LIN {X 0,Y 377.924,Z 388.108,A -85,B 0,C 180,E1 -14679.457,E2 -14679.457} C_VEL
LIN {X 0,Y 374.794,Z 386.154,A -85,B 0,C 180,E1 -14680.722,E2 -14680.722} C_VEL
LIN {X 0,Y 371.596,Z 383.295,A -85,B 0,C 180,E1 -14681.935,E2 -14681.935} C_VEL
LIN {X 0,Y 368.955,Z 380.545,A -85,B 0,C 180,E1 -14682.86,E2 -14682.86} C_VEL
LIN {X 0,Y 365.594,Z 377.85,A -85,B 0,C 180,E1 -14683.883,E2 -14683.883} C_VEL
LIN {X 0,Y 361.342,Z 373.442,A -85,B 0,C 180,E1 -14685.107,E2 -14685.107} C_VEL
LIN {X 0,Y 357.377,Z 369.827,A -85,B 0,C 180,E1 -14686.133,E2 -14686.133} C_VEL
LIN {X 0,Y 354.406,Z 366.631,A -85,B 0,C 180,E1 -14686.847,E2 -14686.847} C_VEL
LIN {X 0,Y 350.901,Z 363.042,A -85,B 0,C 180,E1 -14687.655,E2 -14687.655} C_VEL
LIN {X 0,Y 348.553,Z 360.395,A -85,B 0,C 180,E1 -14688.184,E2 -14688.184} C_VEL
LIN {X 0,Y 345.155,Z 356.37,A -85,B 0,C 180,E1 -14688.921,E2 -14688.921} C_VEL
LIN {X 0,Y 341.007,Z 351.456,A -85,B 0,C 180,E1 -14689.766,E2 -14689.766} C_VEL
LIN {X 0,Y 339.565,Z 349.602,A -85,B 0,C 180,E1 -14690.055,E2 -14690.055} C_VEL
LIN {X 0,Y 337.185,Z 346.417,A -85,B 0,C 180,E1 -14690.522,E2 -14690.522} C_VEL
LIN {X 0,Y 336.133,Z 344.943,A -85,B 0,C 180,E1 -14690.724,E2 -14690.724} C_VEL
LIN {X 0,Y 334.263,Z 342.48,A -85,B 0,C 180,E1 -14691.08,E2 -14691.08} C_VEL
LIN {X 0,Y 333.682,Z 340.419,A -85,B 0,C 180,E1 -14691.257,E2 -14691.257} C_VEL
LIN {X 0,Y 333.715,Z 340.414,A -85,B 0,C 180,E1 -14695.101,E2 -14695.101} C_VEL
LIN {X 0,Y 333.717,Z 340.415,A -85,B 0,C 180,E1 -14697.811,E2 -14697.811} C_VEL
LIN {X 0,Y 333.693,Z 340.421,A -85,B 0,C 180,E1 -14700.362,E2 -14700.362} C_VEL
LIN {X 0,Y 333.67,Z 340.42,A -85,B 0,C 180,E1 -14704.659,E2 -14704.659} C_VEL
LIN {X 0,Y 333.652,Z 340.423,A -85,B 0,C 180,E1 -14707.651,E2 -14707.651} C_VEL
LIN {X 0,Y 333.652,Z 340.421,A -85,B 0,C 180,E1 -14710.766,E2 -14710.766} C_VEL
LIN {X 0,Y 333.659,Z 340.422,A -85,B 0,C 180,E1 -14714.263,E2 -14714.263} C_VEL
LIN {X 0,Y 333.693,Z 340.419,A -85,B 0,C 180,E1 -14717.627,E2 -14717.627} C_VEL
LIN {X 0,Y 333.679,Z 340.419,A -85,B 0,C 180,E1 -14721.196,E2 -14721.196} C_VEL
LIN {X 0,Y 333.682,Z 340.419,A -85,B 0,C 180,E1 -14725.226,E2 -14725.226} C_VEL
LIN {X 0,Y 333.631,Z 340.424,A -85,B 0,C 180,E1 -14728.223,E2 -14728.223} C_VEL
LIN {X 0,Y 333.708,Z 340.415,A -85,B 0,C 180,E1 -14731.029,E2 -14731.029} C_VEL
LIN {X 0,Y 333.709,Z 340.413,A -85,B 0,C 180,E1 -14734.677,E2 -14734.677} C_VEL
LIN {X 0,Y 333.662,Z 340.421,A -85,B 0,C 180,E1 -14737.938,E2 -14737.938} C_VEL
LIN {X 0,Y 333.696,Z 340.413,A -85,B 0,C 180,E1 -14739.91,E2 -14739.91} C_VEL
LIN {X 0,Y 333.087,Z 340.494,A -85,B 0,C 180,E1 -14740.917,E2 -14740.917} C_VEL
LIN {X 0,Y 330.266,Z 340.846,A -85,B 0,C 180,E1 -14742.557,E2 -14742.557} C_VEL
LIN {X 0,Y 327.852,Z 341.148,A -85,B 0,C 180,E1 -14743.884,E2 -14743.884} C_VEL
LIN {X 0,Y 326.829,Z 341.275,A -85,B 0,C 180,E1 -14744.912,E2 -14744.912} C_VEL
LIN {X 0,Y 326.756,Z 341.283,A -85,B 0,C 180,E1 -14745.26,E2 -14745.26} C_VEL
LIN {X 0,Y 326.768,Z 341.282,A -85,B 0,C 180,E1 -14748.84,E2 -14748.84} C_VEL
LIN {X 0,Y 326.965,Z 341.256,A -85,B 0,C 180,E1 -14752.591,E2 -14752.591} C_VEL
LIN {X 0,Y 326.775,Z 341.28,A -85,B 0,C 180,E1 -14755.066,E2 -14755.066} C_VEL
LIN {X 0,Y 327.047,Z 341.239,A -85,B 0,C 180,E1 -14757.537,E2 -14757.537} C_VEL
LIN {X 0,Y 327.178,Z 341.224,A -85,B 0,C 180,E1 -14760.001,E2 -14760.001} C_VEL
LIN {X 0,Y 327.046,Z 341.246,A -85,B 0,C 180,E1 -14762.464,E2 -14762.464} C_VEL
LIN {X 0,Y 326.989,Z 341.252,A -85,B 0,C 180,E1 -14766.17,E2 -14766.17} C_VEL
LIN {X 0,Y 326.914,Z 341.266,A -85,B 0,C 180,E1 -14768.656,E2 -14768.656} C_VEL
LIN {X 0,Y 326.735,Z 341.288,A -85,B 0,C 180,E1 -14772.422,E2 -14772.422} C_VEL
LIN {X 0,Y 326.751,Z 341.283,A -85,B 0,C 180,E1 -14774.958,E2 -14774.958} C_VEL
LIN {X 0,Y 326.707,Z 341.288,A -85,B 0,C 180,E1 -14778.825,E2 -14778.825} C_VEL
LIN {X 0,Y 326.603,Z 341.301,A -85,B 0,C 180,E1 -14782.789,E2 -14782.789} C_VEL
LIN {X 0,Y 326.69,Z 341.29,A -85,B 0,C 180,E1 -14785.484,E2 -14785.484} C_VEL
LIN {X 0,Y 326.649,Z 341.296,A -85,B 0,C 180,E1 -14789.661,E2 -14789.661} C_VEL
LIN {X 0,Y 326.608,Z 341.305,A -85,B 0,C 180,E1 -14794.02,E2 -14794.02} C_VEL
LIN {X 0,Y 326.687,Z 341.65,A -85,B 0,C 180,E1 -14795.511,E2 -14795.511} C_VEL
LIN {X 0,Y 327.029,Z 344.299,A -85,B 0,C 180,E1 -14799.317,E2 -14799.317} C_VEL
LIN {X 0,Y 327.299,Z 346.11,A -85,B 0,C 180,E1 -14801.733,E2 -14801.733} C_VEL
LIN {X 0,Y 327.621,Z 348.814,A -85,B 0,C 180,E1 -14805.065,E2 -14805.065} C_VEL
LIN {X 0,Y 327.642,Z 351.691,A -85,B 0,C 180,E1 -14808.321,E2 -14808.321} C_VEL
LIN {X 0,Y 327.31,Z 354.713,A -85,B 0,C 180,E1 -14811.488,E2 -14811.488} C_VEL
LIN {X 0,Y 326.873,Z 358.059,A -85,B 0,C 180,E1 -14814.789,E2 -14814.789} C_VEL
LIN {X 0,Y 326.311,Z 362.418,A -85,B 0,C 180,E1 -14818.875,E2 -14818.875} C_VEL
LIN {X 0,Y 325.741,Z 367.11,A -85,B 0,C 180,E1 -14823.058,E2 -14823.058} C_VEL
LIN {X 0,Y 325.501,Z 370.259,A -85,B 0,C 180,E1 -14825.781,E2 -14825.781} C_VEL
LIN {X 0,Y 325.309,Z 372.458,A -85,B 0,C 180,E1 -14827.662,E2 -14827.662} C_VEL
LIN {X 0,Y 327.608,Z 381.986,A -85,B 0,C 180,E1 -14828.208,E2 -14828.208} C_VEL
LIN {X 0,Y 329.54,Z 391.658,A -85,B 0,C 180,E1 -14828.869,E2 -14828.869} C_VEL
LIN {X 0,Y 331.098,Z 401.655,A -85,B 0,C 180,E1 -14829.682,E2 -14829.682} C_VEL
LIN {X 0,Y 332.08,Z 410.585,A -85,B 0,C 180,E1 -14830.529,E2 -14830.529} C_VEL
LIN {X 0,Y 332.142,Z 415.477,A -85,B 0,C 180,E1 -14831.015,E2 -14831.015} C_VEL
LIN {X 0,Y 330.814,Z 426.057,A -85,B 0,C 180,E1 -14832.218,E2 -14832.218} C_VEL
LIN {X 0,Y 329.765,Z 433.805,A -85,B 0,C 180,E1 -14833.28,E2 -14833.28} C_VEL
LIN {X 0,Y 328.782,Z 441.599,A -85,B 0,C 180,E1 -14834.558,E2 -14834.558} C_VEL
LIN {X 0,Y 327.797,Z 449.147,A -85,B 0,C 180,E1 -14836.043,E2 -14836.043} C_VEL
LIN {X 0,Y 326.792,Z 455.682,A -85,B 0,C 180,E1 -14837.581,E2 -14837.581} C_VEL
LIN {X 0,Y 326.227,Z 460.185,A -85,B 0,C 180,E1 -14838.82,E2 -14838.82} C_VEL
LIN {X 0,Y 325.599,Z 465.679,A -85,B 0,C 180,E1 -14840.684,E2 -14840.684} C_VEL
LIN {X 0,Y 325.159,Z 470.005,A -85,B 0,C 180,E1 -14842.549,E2 -14842.549} C_VEL
LIN {X 0,Y 324.931,Z 473.023,A -85,B 0,C 180,E1 -14844.241,E2 -14844.241} C_VEL
LIN {X 0,Y 324.902,Z 475.563,A -85,B 0,C 180,E1 -14846.279,E2 -14846.279} C_VEL
LIN {X 0,Y 324.837,Z 476.621,A -85,B 0,C 180,E1 -14847.52,E2 -14847.52} C_VEL
LIN {X 0,Y 324.822,Z 477.21,A -85,B 0,C 180,E1 -14848.76,E2 -14848.76} C_VEL
LIN {X 0,Y 324.873,Z 477.366,A -85,B 0,C 180,E1 -14850,E2 -14850} C_VEL
LIN {X 0,Y 324.822,Z 477.21,A -85,B 0,C 180,E1 -14851.24,E2 -14851.24} C_VEL
LIN {X 0,Y 324.837,Z 476.621,A -85,B 0,C 180,E1 -14852.48,E2 -14852.48} C_VEL
LIN {X 0,Y 324.891,Z 474.173,A -85,B 0,C 180,E1 -14854.964,E2 -14854.964} C_VEL
LIN {X 0,Y 325.047,Z 471.222,A -85,B 0,C 180,E1 -14856.83,E2 -14856.83} C_VEL
LIN {X 0,Y 325.422,Z 467.233,A -85,B 0,C 180,E1 -14858.695,E2 -14858.695} C_VEL
LIN {X 0,Y 325.989,Z 462.102,A -85,B 0,C 180,E1 -14860.559,E2 -14860.559} C_VEL
LIN {X 0,Y 326.645,Z 456.838,A -85,B 0,C 180,E1 -14862.109,E2 -14862.109} C_VEL
LIN {X 0,Y 327.573,Z 450.522,A -85,B 0,C 180,E1 -14863.651,E2 -14863.651} C_VEL
LIN {X 0,Y 328.344,Z 444.569,A -85,B 0,C 180,E1 -14864.883,E2 -14864.883} C_VEL
LIN {X 0,Y 329.294,Z 437.252,A -85,B 0,C 180,E1 -14866.173,E2 -14866.173} C_VEL
LIN {X 0,Y 330.301,Z 429.459,A -85,B 0,C 180,E1 -14867.331,E2 -14867.331} C_VEL
LIN {X 0,Y 331.446,Z 420.95,A -85,B 0,C 180,E1 -14868.385,E2 -14868.385} C_VEL
LIN {X 0,Y 332.274,Z 413.865,A -85,B 0,C 180,E1 -14869.138,E2 -14869.138} C_VEL
LIN {X 0,Y 331.357,Z 403.647,A -85,B 0,C 180,E1 -14870.143,E2 -14870.143} C_VEL
LIN {X 0,Y 329.897,Z 393.628,A -85,B 0,C 180,E1 -14870.983,E2 -14870.983} C_VEL
LIN {X 0,Y 327.918,Z 383.353,A -85,B 0,C 180,E1 -14871.706,E2 -14871.706} C_VEL
LIN {X 0,Y 325.314,Z 372.455,A -85,B 0,C 180,E1 -14872.34,E2 -14872.34} C_VEL
LIN {X 0,Y 325.592,Z 368.677,A -85,B 0,C 180,E1 -14875.576,E2 -14875.576} C_VEL
LIN {X 0,Y 325.918,Z 365.533,A -85,B 0,C 180,E1 -14878.32,E2 -14878.32} C_VEL
LIN {X 0,Y 326.311,Z 362.417,A -85,B 0,C 180,E1 -14881.125,E2 -14881.125} C_VEL
LIN {X 0,Y 326.697,Z 359.315,A -85,B 0,C 180,E1 -14884.009,E2 -14884.009} C_VEL
LIN {X 0,Y 327.166,Z 355.855,A -85,B 0,C 180,E1 -14887.361,E2 -14887.361} C_VEL
LIN {X 0,Y 327.489,Z 353.181,A -85,B 0,C 180,E1 -14890.076,E2 -14890.076} C_VEL
LIN {X 0,Y 327.673,Z 350.303,A -85,B 0,C 180,E1 -14893.176,E2 -14893.176} C_VEL
LIN {X 0,Y 327.615,Z 348.669,A -85,B 0,C 180,E1 -14895.065,E2 -14895.065} C_VEL
LIN {X 0,Y 327.24,Z 345.695,A -85,B 0,C 180,E1 -14898.736,E2 -14898.736} C_VEL
LIN {X 0,Y 326.821,Z 342.844,A -85,B 0,C 180,E1 -14902.716,E2 -14902.716} C_VEL
LIN {X 0,Y 326.64,Z 341.425,A -85,B 0,C 180,E1 -14904.846,E2 -14904.846} C_VEL
LIN {X 0,Y 326.609,Z 341.304,A -85,B 0,C 180,E1 -14907.455,E2 -14907.455} C_VEL
LIN {X 0,Y 326.649,Z 341.296,A -85,B 0,C 180,E1 -14910.339,E2 -14910.339} C_VEL
LIN {X 0,Y 326.69,Z 341.289,A -85,B 0,C 180,E1 -14914.516,E2 -14914.516} C_VEL
LIN {X 0,Y 326.618,Z 341.298,A -85,B 0,C 180,E1 -14918.543,E2 -14918.543} C_VEL
LIN {X 0,Y 326.707,Z 341.288,A -85,B 0,C 180,E1 -14921.175,E2 -14921.175} C_VEL
LIN {X 0,Y 326.763,Z 341.284,A -85,B 0,C 180,E1 -14925.433,E2 -14925.433} C_VEL
LIN {X 0,Y 326.77,Z 341.279,A -85,B 0,C 180,E1 -14928.838,E2 -14928.838} C_VEL
LIN {X 0,Y 326.966,Z 341.254,A -85,B 0,C 180,E1 -14932.589,E2 -14932.589} C_VEL
LIN {X 0,Y 326.775,Z 341.281,A -85,B 0,C 180,E1 -14935.064,E2 -14935.064} C_VEL
LIN {X 0,Y 327.046,Z 341.246,A -85,B 0,C 180,E1 -14937.536,E2 -14937.536} C_VEL
LIN {X 0,Y 327.178,Z 341.224,A -85,B 0,C 180,E1 -14939.999,E2 -14939.999} C_VEL
LIN {X 0,Y 327.047,Z 341.239,A -85,B 0,C 180,E1 -14942.463,E2 -14942.463} C_VEL
LIN {X 0,Y 326.964,Z 341.253,A -85,B 0,C 180,E1 -14946.579,E2 -14946.579} C_VEL
LIN {X 0,Y 326.913,Z 341.263,A -85,B 0,C 180,E1 -14948.654,E2 -14948.654} C_VEL
LIN {X 0,Y 326.733,Z 341.285,A -85,B 0,C 180,E1 -14952.421,E2 -14952.421} C_VEL
LIN {X 0,Y 326.752,Z 341.284,A -85,B 0,C 180,E1 -14954.957,E2 -14954.957} C_VEL
LIN {X 0,Y 326.73,Z 341.286,A -85,B 0,C 180,E1 -14958.837,E2 -14958.837} C_VEL
LIN {X 0,Y 326.601,Z 341.303,A -85,B 0,C 180,E1 -14962.788,E2 -14962.788} C_VEL
LIN {X 0,Y 326.687,Z 341.288,A -85,B 0,C 180,E1 -14965.483,E2 -14965.483} C_VEL
LIN {X 0,Y 326.658,Z 341.292,A -85,B 0,C 180,E1 -14969.658,E2 -14969.658} C_VEL
LIN {X 0,Y 326.605,Z 341.301,A -85,B 0,C 180,E1 -14974.019,E2 -14974.019} C_VEL
LIN {X 0,Y 326.626,Z 341.296,A -85,B 0,C 180,E1 -14977.239,E2 -14977.239} C_VEL
LIN {X 0,Y 326.632,Z 341.301,A -85,B 0,C 180,E1 -14980.202,E2 -14980.202} C_VEL
LIN {X 0,Y 326.626,Z 341.297,A -85,B 0,C 180,E1 -14983.514,E2 -14983.514} C_VEL
LIN {X 0,Y 326.614,Z 341.298,A -85,B 0,C 180,E1 -14987.02,E2 -14987.02} C_VEL
LIN {X 0,Y 326.639,Z 341.296,A -85,B 0,C 180,E1 -14991.394,E2 -14991.394} C_VEL
LIN {X 0,Y 326.616,Z 341.298,A -85,B 0,C 180,E1 -14994.851,E2 -14994.851} C_VEL
LIN {X 0,Y 326.606,Z 341.302,A -85,B 0,C 180,E1 -14997.456,E2 -14997.456} C_VEL
LIN {X 0,Y 326.657,Z 341.294,A -85,B 0,C 180,E1 -15000.341,E2 -15000.341} C_VEL
LIN {X 0,Y 326.686,Z 341.29,A -85,B 0,C 180,E1 -15004.516,E2 -15004.516} C_VEL
LIN {X 0,Y 326.69,Z 341.437,A -85,B 0,C 180,E1 -15007.848,E2 -15007.848} C_VEL
LIN {X 0,Y 327.659,Z 344.132,A -85,B 0,C 180,E1 -15008.04,E2 -15008.04} C_VEL
LIN {X 0,Y 329.516,Z 346.658,A -85,B 0,C 180,E1 -15008.363,E2 -15008.363} C_VEL
LIN {X 0,Y 331.952,Z 350.091,A -85,B 0,C 180,E1 -15008.798,E2 -15008.798} C_VEL
LIN {X 0,Y 335.944,Z 355.201,A -85,B 0,C 180,E1 -15009.531,E2 -15009.531} C_VEL
LIN {X 0,Y 340.312,Z 360.5,A -85,B 0,C 180,E1 -15010.382,E2 -15010.382} C_VEL
LIN {X 0,Y 345.277,Z 366.214,A -85,B 0,C 180,E1 -15011.407,E2 -15011.407} C_VEL
LIN {X 0,Y 347.741,Z 368.91,A -85,B 0,C 180,E1 -15011.95,E2 -15011.95} C_VEL
LIN {X 0,Y 351.899,Z 373.108,A -85,B 0,C 180,E1 -15012.9,E2 -15012.9} C_VEL
LIN {X 0,Y 357.064,Z 378.504,A -85,B 0,C 180,E1 -15014.194,E2 -15014.194} C_VEL
LIN {X 0,Y 360.006,Z 381.132,A -85,B 0,C 180,E1 -15014.986,E2 -15014.986} C_VEL
LIN {X 0,Y 364.311,Z 385.486,A -85,B 0,C 180,E1 -15016.266,E2 -15016.266} C_VEL
LIN {X 0,Y 367.461,Z 388.003,A -85,B 0,C 180,E1 -15017.266,E2 -15017.266} C_VEL
LIN {X 0,Y 370.73,Z 391.389,A -85,B 0,C 180,E1 -15018.475,E2 -15018.475} C_VEL
LIN {X 0,Y 372.478,Z 392.765,A -85,B 0,C 180,E1 -15019.124,E2 -15019.124} C_VEL
LIN {X 0,Y 375.437,Z 394.669,A -85,B 0,C 180,E1 -15020.301,E2 -15020.301} C_VEL
LIN {X 0,Y 377.672,Z 397.002,A -85,B 0,C 180,E1 -15021.439,E2 -15021.439} C_VEL
LIN {X 0,Y 379.602,Z 398.958,A -85,B 0,C 180,E1 -15022.554,E2 -15022.554} C_VEL
LIN {X 0,Y 381.671,Z 400.617,A -85,B 0,C 180,E1 -15023.896,E2 -15023.896} C_VEL
LIN {X 0,Y 382.798,Z 401.351,A -85,B 0,C 180,E1 -15024.733,E2 -15024.733} C_VEL
LIN {X 0,Y 384.081,Z 401.881,A -85,B 0,C 180,E1 -15025.803,E2 -15025.803} C_VEL
LIN {X 0,Y 385.11,Z 402.145,A -85,B 0,C 180,E1 -15026.862,E2 -15026.862} C_VEL
LIN {X 0,Y 385.855,Z 402.309,A -85,B 0,C 180,E1 -15027.912,E2 -15027.912} C_VEL
LIN {X 0,Y 386.321,Z 402.381,A -85,B 0,C 180,E1 -15028.958,E2 -15028.958} C_VEL
LIN {X 0,Y 386.476,Z 402.434,A -85,B 0,C 180,E1 -15030,E2 -15030} C_VEL
LIN {X 0,Y 386.321,Z 402.378,A -85,B 0,C 180,E1 -15031.042,E2 -15031.042} C_VEL
LIN {X 0,Y 385.842,Z 402.331,A -85,B 0,C 180,E1 -15032.088,E2 -15032.088} C_VEL
LIN {X 0,Y 385.11,Z 402.131,A -85,B 0,C 180,E1 -15033.138,E2 -15033.138} C_VEL
LIN {X 0,Y 384.081,Z 401.905,A -85,B 0,C 180,E1 -15034.197,E2 -15034.197} C_VEL
LIN {X 0,Y 381.664,Z 400.618,A -85,B 0,C 180,E1 -15036.094,E2 -15036.094} C_VEL
LIN {X 0,Y 379.589,Z 398.944,A -85,B 0,C 180,E1 -15037.447,E2 -15037.447} C_VEL
LIN {X 0,Y 377.029,Z 396.25,A -85,B 0,C 180,E1 -15038.91,E2 -15038.91} C_VEL
LIN {X 0,Y 375.363,Z 394.639,A -85,B 0,C 180,E1 -15039.701,E2 -15039.701} C_VEL
LIN {X 0,Y 372.225,Z 392.625,A -85,B 0,C 180,E1 -15040.947,E2 -15040.947} C_VEL
LIN {X 0,Y 368.356,Z 389.042,A -85,B 0,C 180,E1 -15042.404,E2 -15042.404} C_VEL
LIN {X 0,Y 366.373,Z 387.02,A -85,B 0,C 180,E1 -15043.098,E2 -15043.098} C_VEL
LIN {X 0,Y 362.149,Z 383.496,A -85,B 0,C 180,E1 -15044.376,E2 -15044.376} C_VEL
LIN {X 0,Y 358.454,Z 379.654,A -85,B 0,C 180,E1 -15045.437,E2 -15045.437} C_VEL
LIN {X 0,Y 354.263,Z 375.76,A -85,B 0,C 180,E1 -15046.509,E2 -15046.509} C_VEL
LIN {X 0,Y 351.167,Z 372.459,A -85,B 0,C 180,E1 -15047.265,E2 -15047.265} C_VEL
LIN {X 0,Y 347.177,Z 368.214,A -85,B 0,C 180,E1 -15048.186,E2 -15048.186} C_VEL
LIN {X 0,Y 342.185,Z 362.733,A -85,B 0,C 180,E1 -15049.237,E2 -15049.237} C_VEL
LIN {X 0,Y 339.905,Z 360.102,A -85,B 0,C 180,E1 -15049.698,E2 -15049.698} C_VEL
LIN {X 0,Y 334.964,Z 354.182,A -85,B 0,C 180,E1 -15050.647,E2 -15050.647} C_VEL
LIN {X 0,Y 331.85,Z 350.001,A -85,B 0,C 180,E1 -15051.218,E2 -15051.218} C_VEL
LIN {X 0,Y 329.514,Z 346.635,A -85,B 0,C 180,E1 -15051.636,E2 -15051.636} C_VEL
LIN {X 0,Y 328.327,Z 345.052,A -85,B 0,C 180,E1 -15051.847,E2 -15051.847} C_VEL
LIN {X 0,Y 326.954,Z 342.586,A -85,B 0,C 180,E1 -15052.089,E2 -15052.089} C_VEL
LIN {X 0,Y 326.676,Z 341.295,A -85,B 0,C 180,E1 -15052.178,E2 -15052.178} C_VEL
LIN {X 0,Y 326.686,Z 341.29,A -85,B 0,C 180,E1 -15055.484,E2 -15055.484} C_VEL
LIN {X 0,Y 326.657,Z 341.294,A -85,B 0,C 180,E1 -15059.659,E2 -15059.659} C_VEL
LIN {X 0,Y 326.604,Z 341.303,A -85,B 0,C 180,E1 -15064.02,E2 -15064.02} C_VEL
LIN {X 0,Y 326.626,Z 341.297,A -85,B 0,C 180,E1 -15067.239,E2 -15067.239} C_VEL
LIN {X 0,Y 326.6,Z 341.303,A -85,B 0,C 180,E1 -15070.207,E2 -15070.207} C_VEL
LIN {X 0,Y 326.607,Z 341.3,A -85,B 0,C 180,E1 -15073.518,E2 -15073.518} C_VEL
LIN {X 0,Y 326.629,Z 341.296,A -85,B 0,C 180,E1 -15077.018,E2 -15077.018} C_VEL
LIN {X 0,Y 326.642,Z 341.294,A -85,B 0,C 180,E1 -15080.766,E2 -15080.766} C_VEL
LIN {X 0,Y 326.609,Z 341.298,A -85,B 0,C 180,E1 -15084.481,E2 -15084.481} C_VEL
LIN {X 0,Y 326.607,Z 341.302,A -85,B 0,C 180,E1 -15087.456,E2 -15087.456} C_VEL
LIN {X 0,Y 326.658,Z 341.292,A -85,B 0,C 180,E1 -15090.342,E2 -15090.342} C_VEL
LIN {X 0,Y 326.687,Z 341.288,A -85,B 0,C 180,E1 -15094.517,E2 -15094.517} C_VEL
LIN {X 0,Y 326.618,Z 341.297,A -85,B 0,C 180,E1 -15098.544,E2 -15098.544} C_VEL
LIN {X 0,Y 326.742,Z 341.285,A -85,B 0,C 180,E1 -15101.178,E2 -15101.178} C_VEL
LIN {X 0,Y 326.756,Z 341.283,A -85,B 0,C 180,E1 -15105.26,E2 -15105.26} C_VEL
LIN {X 0,Y 326.105,Z 341.362,A -85,B 0,C 180,E1 -15106.289,E2 -15106.289} C_VEL
LIN {X 0,Y 323.24,Z 341.718,A -85,B 0,C 180,E1 -15107.964,E2 -15107.964} C_VEL
LIN {X 0,Y 320.833,Z 342.02,A -85,B 0,C 180,E1 -15109.321,E2 -15109.321} C_VEL
LIN {X 0,Y 319.849,Z 342.14,A -85,B 0,C 180,E1 -15110.371,E2 -15110.371} C_VEL
LIN {X 0,Y 319.795,Z 342.147,A -85,B 0,C 180,E1 -15110.727,E2 -15110.727} C_VEL
LIN {X 0,Y 319.944,Z 342.129,A -85,B 0,C 180,E1 -15113.695,E2 -15113.695} C_VEL
LIN {X 0,Y 319.99,Z 342.117,A -85,B 0,C 180,E1 -15117.483,E2 -15117.483} C_VEL
LIN {X 0,Y 320.131,Z 342.102,A -85,B 0,C 180,E1 -15120.001,E2 -15120.001} C_VEL
LIN {X 0,Y 319.99,Z 342.125,A -85,B 0,C 180,E1 -15122.518,E2 -15122.518} C_VEL
LIN {X 0,Y 319.944,Z 342.131,A -85,B 0,C 180,E1 -15126.306,E2 -15126.306} C_VEL
LIN {X 0,Y 319.842,Z 342.145,A -85,B 0,C 180,E1 -15128.849,E2 -15128.849} C_VEL
LIN {X 0,Y 319.683,Z 342.166,A -85,B 0,C 180,E1 -15132.7,E2 -15132.7} C_VEL
LIN {X 0,Y 319.679,Z 342.162,A -85,B 0,C 180,E1 -15135.297,E2 -15135.297} C_VEL
LIN {X 0,Y 319.629,Z 342.168,A -85,B 0,C 180,E1 -15139.259,E2 -15139.259} C_VEL
LIN {X 0,Y 319.561,Z 342.177,A -85,B 0,C 180,E1 -15143.321,E2 -15143.321} C_VEL
LIN {X 0,Y 319.635,Z 342.173,A -85,B 0,C 180,E1 -15146.089,E2 -15146.089} C_VEL
LIN {X 0,Y 319.581,Z 342.175,A -85,B 0,C 180,E1 -15148.935,E2 -15148.935} C_VEL
LIN {X 0,Y 319.531,Z 342.186,A -85,B 0,C 180,E1 -15151.863,E2 -15151.863} C_VEL
LIN {X 0,Y 319.589,Z 342.373,A -85,B 0,C 180,E1 -15154.874,E2 -15154.874} C_VEL
LIN {X 0,Y 319.872,Z 344.413,A -85,B 0,C 180,E1 -15157.967,E2 -15157.967} C_VEL
LIN {X 0,Y 320.294,Z 347.157,A -85,B 0,C 180,E1 -15161.752,E2 -15161.752} C_VEL
LIN {X 0,Y 320.586,Z 350.124,A -85,B 0,C 180,E1 -15165.452,E2 -15165.452} C_VEL
LIN {X 0,Y 320.556,Z 353.125,A -85,B 0,C 180,E1 -15168.873,E2 -15168.873} C_VEL
LIN {X 0,Y 320.165,Z 356.28,A -85,B 0,C 180,E1 -15172.209,E2 -15172.209} C_VEL
LIN {X 0,Y 319.739,Z 359.2,A -85,B 0,C 180,E1 -15175.146,E2 -15175.146} C_VEL
LIN {X 0,Y 319.179,Z 363.848,A -85,B 0,C 180,E1 -15179.573,E2 -15179.573} C_VEL
LIN {X 0,Y 318.563,Z 368.537,A -85,B 0,C 180,E1 -15183.818,E2 -15183.818} C_VEL
LIN {X 0,Y 318.267,Z 372.29,A -85,B 0,C 180,E1 -15187.142,E2 -15187.142} C_VEL
LIN {X 0,Y 320.637,Z 382.141,A -85,B 0,C 180,E1 -15187.727,E2 -15187.727} C_VEL
LIN {X 0,Y 322.644,Z 391.623,A -85,B 0,C 180,E1 -15188.406,E2 -15188.406} C_VEL
LIN {X 0,Y 324.102,Z 400.876,A -85,B 0,C 180,E1 -15189.176,E2 -15189.176} C_VEL
LIN {X 0,Y 325.141,Z 410.382,A -85,B 0,C 180,E1 -15190.096,E2 -15190.096} C_VEL
LIN {X 0,Y 325.408,Z 415.28,A -85,B 0,C 180,E1 -15190.606,E2 -15190.606} C_VEL
LIN {X 0,Y 324.026,Z 425.86,A -85,B 0,C 180,E1 -15191.833,E2 -15191.833} C_VEL
LIN {X 0,Y 322.946,Z 433.605,A -85,B 0,C 180,E1 -15192.915,E2 -15192.915} C_VEL
LIN {X 0,Y 321.873,Z 441.733,A -85,B 0,C 180,E1 -15194.284,E2 -15194.284} C_VEL
LIN {X 0,Y 320.898,Z 448.951,A -85,B 0,C 180,E1 -15195.736,E2 -15195.736} C_VEL
LIN {X 0,Y 319.842,Z 455.486,A -85,B 0,C 180,E1 -15197.307,E2 -15197.307} C_VEL
LIN {X 0,Y 319.218,Z 459.988,A -85,B 0,C 180,E1 -15198.571,E2 -15198.571} C_VEL
LIN {X 0,Y 318.562,Z 465.482,A -85,B 0,C 180,E1 -15200.476,E2 -15200.476} C_VEL
LIN {X 0,Y 318.087,Z 469.808,A -85,B 0,C 180,E1 -15202.382,E2 -15202.382} C_VEL
LIN {X 0,Y 317.847,Z 473.062,A -85,B 0,C 180,E1 -15204.278,E2 -15204.278} C_VEL
LIN {X 0,Y 317.81,Z 475.367,A -85,B 0,C 180,E1 -15206.196,E2 -15206.196} C_VEL
LIN {X 0,Y 317.759,Z 476.426,A -85,B 0,C 180,E1 -15207.465,E2 -15207.465} C_VEL
LIN {X 0,Y 317.734,Z 477.014,A -85,B 0,C 180,E1 -15208.733,E2 -15208.733} C_VEL
LIN {X 0,Y 317.734,Z 477.014,A -85,B 0,C 180,E1 -15211.267,E2 -15211.267} C_VEL
LIN {X 0,Y 317.759,Z 476.426,A -85,B 0,C 180,E1 -15212.535,E2 -15212.535} C_VEL
LIN {X 0,Y 317.805,Z 473.977,A -85,B 0,C 180,E1 -15215.075,E2 -15215.075} C_VEL
LIN {X 0,Y 317.986,Z 471.026,A -85,B 0,C 180,E1 -15216.982,E2 -15216.982} C_VEL
LIN {X 0,Y 318.381,Z 467.037,A -85,B 0,C 180,E1 -15218.889,E2 -15218.889} C_VEL
LIN {X 0,Y 318.975,Z 461.905,A -85,B 0,C 180,E1 -15220.794,E2 -15220.794} C_VEL
LIN {X 0,Y 319.656,Z 456.641,A -85,B 0,C 180,E1 -15222.378,E2 -15222.378} C_VEL
LIN {X 0,Y 320.669,Z 450.326,A -85,B 0,C 180,E1 -15223.95,E2 -15223.95} C_VEL
LIN {X 0,Y 321.46,Z 444.372,A -85,B 0,C 180,E1 -15225.21,E2 -15225.21} C_VEL
LIN {X 0,Y 322.408,Z 437.444,A -85,B 0,C 180,E1 -15226.462,E2 -15226.462} C_VEL
LIN {X 0,Y 323.505,Z 429.263,A -85,B 0,C 180,E1 -15227.707,E2 -15227.707} C_VEL
LIN {X 0,Y 324.692,Z 420.753,A -85,B 0,C 180,E1 -15228.782,E2 -15228.782} C_VEL
LIN {X 0,Y 325.417,Z 413.665,A -85,B 0,C 180,E1 -15229.557,E2 -15229.557} C_VEL
LIN {X 0,Y 324.427,Z 403.443,A -85,B 0,C 180,E1 -15230.592,E2 -15230.592} C_VEL
LIN {X 0,Y 322.831,Z 392.685,A -85,B 0,C 180,E1 -15231.512,E2 -15231.512} C_VEL
LIN {X 0,Y 320.823,Z 382.682,A -85,B 0,C 180,E1 -15232.234,E2 -15232.234} C_VEL
LIN {X 0,Y 318.267,Z 372.289,A -85,B 0,C 180,E1 -15232.859,E2 -15232.859} C_VEL
LIN {X 0,Y 318.57,Z 368.514,A -85,B 0,C 180,E1 -15236.182,E2 -15236.182} C_VEL
LIN {X 0,Y 318.938,Z 365.397,A -85,B 0,C 180,E1 -15238.998,E2 -15238.998} C_VEL
LIN {X 0,Y 319.34,Z 362.284,A -85,B 0,C 180,E1 -15241.883,E2 -15241.883} C_VEL
LIN {X 0,Y 319.851,Z 358.431,A -85,B 0,C 180,E1 -15245.61,E2 -15245.61} C_VEL
LIN {X 0,Y 320.176,Z 356.134,A -85,B 0,C 180,E1 -15247.923,E2 -15247.923} C_VEL
LIN {X 0,Y 320.547,Z 353.088,A -85,B 0,C 180,E1 -15251.128,E2 -15251.128} C_VEL
LIN {X 0,Y 320.59,Z 350.09,A -85,B 0,C 180,E1 -15254.548,E2 -15254.548} C_VEL
LIN {X 0,Y 320.282,Z 347.144,A -85,B 0,C 180,E1 -15258.251,E2 -15258.251} C_VEL
LIN {X 0,Y 319.87,Z 344.412,A -85,B 0,C 180,E1 -15262.033,E2 -15262.033} C_VEL
LIN {X 0,Y 319.589,Z 342.375,A -85,B 0,C 180,E1 -15265.126,E2 -15265.126} C_VEL
LIN {X 0,Y 319.531,Z 342.187,A -85,B 0,C 180,E1 -15268.137,E2 -15268.137} C_VEL
LIN {X 0,Y 319.612,Z 342.174,A -85,B 0,C 180,E1 -15271.59,E2 -15271.59} C_VEL
LIN {X 0,Y 319.603,Z 342.173,A -85,B 0,C 180,E1 -15275.303,E2 -15275.303} C_VEL
LIN {X 0,Y 319.587,Z 342.177,A -85,B 0,C 180,E1 -15279.399,E2 -15279.399} C_VEL
LIN {X 0,Y 319.624,Z 342.17,A -85,B 0,C 180,E1 -15282.07,E2 -15282.07} C_VEL
LIN {X 0,Y 319.732,Z 342.157,A -85,B 0,C 180,E1 -15286.007,E2 -15286.007} C_VEL
LIN {X 0,Y 319.757,Z 342.154,A -85,B 0,C 180,E1 -15289.872,E2 -15289.872} C_VEL
LIN {X 0,Y 319.925,Z 342.131,A -85,B 0,C 180,E1 -15292.425,E2 -15292.425} C_VEL
LIN {X 0,Y 319.745,Z 342.156,A -85,B 0,C 180,E1 -15294.955,E2 -15294.955} C_VEL
LIN {X 0,Y 319.99,Z 342.125,A -85,B 0,C 180,E1 -15297.482,E2 -15297.482} C_VEL
LIN {X 0,Y 320.131,Z 342.102,A -85,B 0,C 180,E1 -15299.999,E2 -15299.999} C_VEL
LIN {X 0,Y 319.99,Z 342.117,A -85,B 0,C 180,E1 -15302.517,E2 -15302.517} C_VEL
LIN {X 0,Y 319.927,Z 342.129,A -85,B 0,C 180,E1 -15306.567,E2 -15306.567} C_VEL
LIN {X 0,Y 319.841,Z 342.146,A -85,B 0,C 180,E1 -15308.847,E2 -15308.847} C_VEL
LIN {X 0,Y 319.681,Z 342.165,A -85,B 0,C 180,E1 -15312.699,E2 -15312.699} C_VEL
LIN {X 0,Y 319.698,Z 342.16,A -85,B 0,C 180,E1 -15315.295,E2 -15315.295} C_VEL
LIN {X 0,Y 319.672,Z 342.162,A -85,B 0,C 180,E1 -15319.254,E2 -15319.254} C_VEL
LIN {X 0,Y 319.558,Z 342.177,A -85,B 0,C 180,E1 -15323.32,E2 -15323.32} C_VEL
LIN {X 0,Y 319.632,Z 342.168,A -85,B 0,C 180,E1 -15326.087,E2 -15326.087} C_VEL
LIN {X 0,Y 319.587,Z 342.175,A -85,B 0,C 180,E1 -15328.933,E2 -15328.933} C_VEL
LIN {X 0,Y 319.531,Z 342.181,A -85,B 0,C 180,E1 -15331.861,E2 -15331.861} C_VEL
LIN {X 0,Y 319.577,Z 342.175,A -85,B 0,C 180,E1 -15335.543,E2 -15335.543} C_VEL
LIN {X 0,Y 319.596,Z 342.175,A -85,B 0,C 180,E1 -15338.004,E2 -15338.004} C_VEL
LIN {X 0,Y 319.594,Z 342.173,A -85,B 0,C 180,E1 -15341.611,E2 -15341.611} C_VEL
LIN {X 0,Y 319.578,Z 342.174,A -85,B 0,C 180,E1 -15345.273,E2 -15345.273} C_VEL
LIN {X 0,Y 319.543,Z 342.179,A -85,B 0,C 180,E1 -15348.714,E2 -15348.714} C_VEL
LIN {X 0,Y 319.594,Z 342.174,A -85,B 0,C 180,E1 -15352.339,E2 -15352.339} C_VEL
LIN {X 0,Y 319.556,Z 342.178,A -85,B 0,C 180,E1 -15355.123,E2 -15355.123} C_VEL
LIN {X 0,Y 319.566,Z 342.177,A -85,B 0,C 180,E1 -15359.058,E2 -15359.058} C_VEL
LIN {X 0,Y 319.605,Z 342.172,A -85,B 0,C 180,E1 -15362.498,E2 -15362.498} C_VEL
LIN {X 0,Y 319.601,Z 342.175,A -85,B 0,C 180,E1 -15365.304,E2 -15365.304} C_VEL
LIN {X 0,Y 319.569,Z 342.178,A -85,B 0,C 180,E1 -15367.016,E2 -15367.016} C_VEL
LIN {X 0,Y 320.698,Z 345.22,A -85,B 0,C 180,E1 -15367.235,E2 -15367.235} C_VEL
LIN {X 0,Y 322.178,Z 347.383,A -85,B 0,C 180,E1 -15367.456,E2 -15367.456} C_VEL
LIN {X 0,Y 327.334,Z 354.823,A -85,B 0,C 180,E1 -15368.295,E2 -15368.295} C_VEL
LIN {X 0,Y 332.297,Z 360.963,A -85,B 0,C 180,E1 -15369.178,E2 -15369.178} C_VEL
LIN {X 0,Y 336.801,Z 366.347,A -85,B 0,C 180,E1 -15370.043,E2 -15370.043} C_VEL
LIN {X 0,Y 341.771,Z 372.016,A -85,B 0,C 180,E1 -15371.068,E2 -15371.068} C_VEL
LIN {X 0,Y 347.333,Z 378.066,A -85,B 0,C 180,E1 -15372.331,E2 -15372.331} C_VEL
LIN {X 0,Y 350.394,Z 381.136,A -85,B 0,C 180,E1 -15373.063,E2 -15373.063} C_VEL
LIN {X 0,Y 354.735,Z 385.41,A -85,B 0,C 180,E1 -15374.185,E2 -15374.185} C_VEL
LIN {X 0,Y 356.911,Z 387.392,A -85,B 0,C 180,E1 -15374.765,E2 -15374.765} C_VEL
LIN {X 0,Y 361.779,Z 392.195,A -85,B 0,C 180,E1 -15376.239,E2 -15376.239} C_VEL
LIN {X 0,Y 364.7,Z 394.66,A -85,B 0,C 180,E1 -15377.168,E2 -15377.168} C_VEL
LIN {X 0,Y 367.983,Z 397.925,A -85,B 0,C 180,E1 -15378.388,E2 -15378.388} C_VEL
LIN {X 0,Y 372.69,Z 401.205,A -85,B 0,C 180,E1 -15380.229,E2 -15380.229} C_VEL
LIN {X 0,Y 376.096,Z 404.733,A -85,B 0,C 180,E1 -15382.048,E2 -15382.048} C_VEL
LIN {X 0,Y 378.548,Z 406.863,A -85,B 0,C 180,E1 -15383.604,E2 -15383.604} C_VEL
LIN {X 0,Y 380.799,Z 408.183,A -85,B 0,C 180,E1 -15385.279,E2 -15385.279} C_VEL
LIN {X 0,Y 382.437,Z 408.721,A -85,B 0,C 180,E1 -15386.84,E2 -15386.84} C_VEL
LIN {X 0,Y 383.215,Z 408.887,A -85,B 0,C 180,E1 -15387.898,E2 -15387.898} C_VEL
LIN {X 0,Y 383.694,Z 408.967,A -85,B 0,C 180,E1 -15388.95,E2 -15388.95} C_VEL
LIN {X 0,Y 383.856,Z 409.006,A -85,B 0,C 180,E1 -15390,E2 -15390} C_VEL
LIN {X 0,Y 383.694,Z 408.966,A -85,B 0,C 180,E1 -15391.05,E2 -15391.05} C_VEL
LIN {X 0,Y 383.199,Z 408.915,A -85,B 0,C 180,E1 -15392.102,E2 -15392.102} C_VEL
LIN {X 0,Y 382.437,Z 408.715,A -85,B 0,C 180,E1 -15393.16,E2 -15393.16} C_VEL
LIN {X 0,Y 380.795,Z 408.208,A -85,B 0,C 180,E1 -15394.714,E2 -15394.714} C_VEL
LIN {X 0,Y 378.524,Z 406.893,A -85,B 0,C 180,E1 -15396.396,E2 -15396.396} C_VEL
LIN {X 0,Y 376.093,Z 404.737,A -85,B 0,C 180,E1 -15397.949,E2 -15397.949} C_VEL
LIN {X 0,Y 372.658,Z 401.208,A -85,B 0,C 180,E1 -15399.772,E2 -15399.772} C_VEL
LIN {X 0,Y 369.698,Z 399.29,A -85,B 0,C 180,E1 -15400.959,E2 -15400.959} C_VEL
LIN {X 0,Y 366.472,Z 396.528,A -85,B 0,C 180,E1 -15402.178,E2 -15402.178} C_VEL
LIN {X 0,Y 362.851,Z 392.933,A -85,B 0,C 180,E1 -15403.44,E2 -15403.44} C_VEL
LIN {X 0,Y 360.388,Z 391.005,A -85,B 0,C 180,E1 -15404.187,E2 -15404.187} C_VEL
LIN {X 0,Y 355.423,Z 385.924,A -85,B 0,C 180,E1 -15405.641,E2 -15405.641} C_VEL
LIN {X 0,Y 350.894,Z 381.726,A -85,B 0,C 180,E1 -15406.805,E2 -15406.805} C_VEL
LIN {X 0,Y 347.671,Z 378.362,A -85,B 0,C 180,E1 -15407.594,E2 -15407.594} C_VEL
LIN {X 0,Y 343.083,Z 373.299,A -85,B 0,C 180,E1 -15408.654,E2 -15408.654} C_VEL
LIN {X 0,Y 338.496,Z 368.416,A -85,B 0,C 180,E1 -15409.608,E2 -15409.608} C_VEL
LIN {X 0,Y 336.042,Z 365.571,A -85,B 0,C 180,E1 -15410.103,E2 -15410.103} C_VEL
LIN {X 0,Y 329.245,Z 357.244,A -85,B 0,C 180,E1 -15411.373,E2 -15411.373} C_VEL
LIN {X 0,Y 325.098,Z 351.701,A -85,B 0,C 180,E1 -15412.079,E2 -15412.079} C_VEL
LIN {X 0,Y 322.035,Z 347.092,A -85,B 0,C 180,E1 -15412.569,E2 -15412.569} C_VEL
LIN {X 0,Y 319.966,Z 343.736,A -85,B 0,C 180,E1 -15412.879,E2 -15412.879} C_VEL
LIN {X 0,Y 319.571,Z 342.182,A -85,B 0,C 180,E1 -15412.961,E2 -15412.961} C_VEL
LIN {X 0,Y 319.631,Z 342.172,A -85,B 0,C 180,E1 -15416.088,E2 -15416.088} C_VEL
LIN {X 0,Y 319.585,Z 342.175,A -85,B 0,C 180,E1 -15418.934,E2 -15418.934} C_VEL
LIN {X 0,Y 319.529,Z 342.183,A -85,B 0,C 180,E1 -15421.862,E2 -15421.862} C_VEL
LIN {X 0,Y 319.576,Z 342.176,A -85,B 0,C 180,E1 -15425.543,E2 -15425.543} C_VEL
LIN {X 0,Y 319.594,Z 342.177,A -85,B 0,C 180,E1 -15428.005,E2 -15428.005} C_VEL
LIN {X 0,Y 319.568,Z 342.178,A -85,B 0,C 180,E1 -15431.607,E2 -15431.607} C_VEL
LIN {X 0,Y 319.584,Z 342.174,A -85,B 0,C 180,E1 -15435.275,E2 -15435.275} C_VEL
LIN {X 0,Y 319.577,Z 342.174,A -85,B 0,C 180,E1 -15438.72,E2 -15438.72} C_VEL
LIN {X 0,Y 319.595,Z 342.173,A -85,B 0,C 180,E1 -15442.34,E2 -15442.34} C_VEL
LIN {X 0,Y 319.557,Z 342.178,A -85,B 0,C 180,E1 -15445.124,E2 -15445.124} C_VEL
LIN {X 0,Y 319.568,Z 342.177,A -85,B 0,C 180,E1 -15449.058,E2 -15449.058} C_VEL
LIN {X 0,Y 319.606,Z 342.171,A -85,B 0,C 180,E1 -15452.499,E2 -15452.499} C_VEL
LIN {X 0,Y 319.601,Z 342.174,A -85,B 0,C 180,E1 -15455.305,E2 -15455.305} C_VEL
LIN {X 0,Y 319.602,Z 342.174,A -85,B 0,C 180,E1 -15459.401,E2 -15459.401} C_VEL
LIN {X 0,Y 319.656,Z 342.165,A -85,B 0,C 180,E1 -15462.074,E2 -15462.074} C_VEL
LIN {X 0,Y 319.73,Z 342.154,A -85,B 0,C 180,E1 -15466.008,E2 -15466.008} C_VEL
LIN {X 0,Y 319.756,Z 342.151,A -85,B 0,C 180,E1 -15469.874,E2 -15469.874} C_VEL
LIN {X 0,Y 319.795,Z 342.147,A -85,B 0,C 180,E1 -15470.727,E2 -15470.727} C_VEL
LIN {X 0,Y 319.518,Z 342.186,A -85,B 0,C 180,E1 -15471.431,E2 -15471.431} C_VEL
LIN {X 0,Y 317.546,Z 342.437,A -85,B 0,C 180,E1 -15472.809,E2 -15472.809} C_VEL
LIN {X 0,Y 313.745,Z 342.907,A -85,B 0,C 180,E1 -15474.874,E2 -15474.874} C_VEL
LIN {X 0,Y 312.755,Z 343.023,A -85,B 0,C 180,E1 -15475.949,E2 -15475.949} C_VEL
LIN {X 0,Y 312.717,Z 343.025,A -85,B 0,C 180,E1 -15476.313,E2 -15476.313} C_VEL
LIN {X 0,Y 312.988,Z 342.99,A -85,B 0,C 180,E1 -15478.714,E2 -15478.714} C_VEL
LIN {X 0,Y 312.99,Z 342.995,A -85,B 0,C 180,E1 -15481.287,E2 -15481.287} C_VEL
LIN {X 0,Y 312.715,Z 343.031,A -85,B 0,C 180,E1 -15485.158,E2 -15485.158} C_VEL
LIN {X 0,Y 312.866,Z 343.011,A -85,B 0,C 180,E1 -15487.747,E2 -15487.747} C_VEL
LIN {X 0,Y 312.67,Z 343.036,A -85,B 0,C 180,E1 -15491.672,E2 -15491.672} C_VEL
LIN {X 0,Y 312.667,Z 343.038,A -85,B 0,C 180,E1 -15494.866,E2 -15494.866} C_VEL
LIN {X 0,Y 312.586,Z 343.046,A -85,B 0,C 180,E1 -15499.213,E2 -15499.213} C_VEL
LIN {X 0,Y 312.527,Z 343.055,A -85,B 0,C 180,E1 -15502.781,E2 -15502.781} C_VEL
LIN {X 0,Y 312.603,Z 343.048,A -85,B 0,C 180,E1 -15505.936,E2 -15505.936} C_VEL
LIN {X 0,Y 312.539,Z 343.054,A -85,B 0,C 180,E1 -15509.651,E2 -15509.651} C_VEL
LIN {X 0,Y 312.525,Z 343.06,A -85,B 0,C 180,E1 -15513.691,E2 -15513.691} C_VEL
LIN {X 0,Y 312.521,Z 343.092,A -85,B 0,C 180,E1 -15514.209,E2 -15514.209} C_VEL
LIN {X 0,Y 312.863,Z 345.644,A -85,B 0,C 180,E1 -15518.166,E2 -15518.166} C_VEL
LIN {X 0,Y 313.132,Z 347.346,A -85,B 0,C 180,E1 -15520.609,E2 -15520.609} C_VEL
LIN {X 0,Y 313.471,Z 350.05,A -85,B 0,C 180,E1 -15524.157,E2 -15524.157} C_VEL
LIN {X 0,Y 313.569,Z 353.041,A -85,B 0,C 180,E1 -15527.749,E2 -15527.749} C_VEL
LIN {X 0,Y 313.234,Z 356.051,A -85,B 0,C 180,E1 -15531.08,E2 -15531.08} C_VEL
LIN {X 0,Y 312.81,Z 359.084,A -85,B 0,C 180,E1 -15534.257,E2 -15534.257} C_VEL
LIN {X 0,Y 312.192,Z 363.711,A -85,B 0,C 180,E1 -15538.817,E2 -15538.817} C_VEL
LIN {X 0,Y 311.547,Z 368.366,A -85,B 0,C 180,E1 -15543.182,E2 -15543.182} C_VEL
LIN {X 0,Y 311.226,Z 372.263,A -85,B 0,C 180,E1 -15546.605,E2 -15546.605} C_VEL
LIN {X 0,Y 313.726,Z 382.324,A -85,B 0,C 180,E1 -15547.228,E2 -15547.228} C_VEL
LIN {X 0,Y 315.66,Z 391.284,A -85,B 0,C 180,E1 -15547.895,E2 -15547.895} C_VEL
LIN {X 0,Y 317.179,Z 400.839,A -85,B 0,C 180,E1 -15548.713,E2 -15548.713} C_VEL
LIN {X 0,Y 318.254,Z 410.18,A -85,B 0,C 180,E1 -15549.647,E2 -15549.647} C_VEL
LIN {X 0,Y 318.55,Z 416.504,A -85,B 0,C 180,E1 -15550.339,E2 -15550.339} C_VEL
LIN {X 0,Y 317.109,Z 426.798,A -85,B 0,C 180,E1 -15551.59,E2 -15551.59} C_VEL
LIN {X 0,Y 315.848,Z 435.328,A -85,B 0,C 180,E1 -15552.853,E2 -15552.853} C_VEL
LIN {X 0,Y 314.782,Z 443.027,A -85,B 0,C 180,E1 -15554.225,E2 -15554.225} C_VEL
LIN {X 0,Y 313.734,Z 450.129,A -85,B 0,C 180,E1 -15555.735,E2 -15555.735} C_VEL
LIN {X 0,Y 312.692,Z 456.444,A -85,B 0,C 180,E1 -15557.342,E2 -15557.342} C_VEL
LIN {X 0,Y 311.972,Z 461.708,A -85,B 0,C 180,E1 -15558.961,E2 -15558.961} C_VEL
LIN {X 0,Y 311.354,Z 466.84,A -85,B 0,C 180,E1 -15560.909,E2 -15560.909} C_VEL
LIN {X 0,Y 310.925,Z 470.83,A -85,B 0,C 180,E1 -15562.859,E2 -15562.859} C_VEL
LIN {X 0,Y 310.717,Z 473.781,A -85,B 0,C 180,E1 -15564.809,E2 -15564.809} C_VEL
LIN {X 0,Y 310.683,Z 476.23,A -85,B 0,C 180,E1 -15567.407,E2 -15567.407} C_VEL
LIN {X 0,Y 310.649,Z 476.819,A -85,B 0,C 180,E1 -15568.704,E2 -15568.704} C_VEL
LIN {X 0,Y 310.649,Z 476.819,A -85,B 0,C 180,E1 -15571.296,E2 -15571.296} C_VEL
LIN {X 0,Y 310.683,Z 476.23,A -85,B 0,C 180,E1 -15572.593,E2 -15572.593} C_VEL
LIN {X 0,Y 310.708,Z 473.78,A -85,B 0,C 180,E1 -15575.191,E2 -15575.191} C_VEL
LIN {X 0,Y 310.921,Z 470.829,A -85,B 0,C 180,E1 -15577.142,E2 -15577.142} C_VEL
LIN {X 0,Y 311.354,Z 466.84,A -85,B 0,C 180,E1 -15579.091,E2 -15579.091} C_VEL
LIN {X 0,Y 311.972,Z 461.708,A -85,B 0,C 180,E1 -15581.039,E2 -15581.039} C_VEL
LIN {X 0,Y 312.693,Z 456.444,A -85,B 0,C 180,E1 -15582.658,E2 -15582.658} C_VEL
LIN {X 0,Y 313.756,Z 450.13,A -85,B 0,C 180,E1 -15584.264,E2 -15584.264} C_VEL
LIN {X 0,Y 314.793,Z 443.014,A -85,B 0,C 180,E1 -15585.777,E2 -15585.777} C_VEL
LIN {X 0,Y 315.849,Z 435.328,A -85,B 0,C 180,E1 -15587.147,E2 -15587.147} C_VEL
LIN {X 0,Y 317.044,Z 426.797,A -85,B 0,C 180,E1 -15588.414,E2 -15588.414} C_VEL
LIN {X 0,Y 318.548,Z 416.504,A -85,B 0,C 180,E1 -15589.661,E2 -15589.661} C_VEL
LIN {X 0,Y 317.773,Z 405.365,A -85,B 0,C 180,E1 -15590.866,E2 -15590.866} C_VEL
LIN {X 0,Y 316.093,Z 393.647,A -85,B 0,C 180,E1 -15591.917,E2 -15591.917} C_VEL
LIN {X 0,Y 313.98,Z 383.144,A -85,B 0,C 180,E1 -15592.712,E2 -15592.712} C_VEL
LIN {X 0,Y 311.305,Z 372.817,A -85,B 0,C 180,E1 -15593.371,E2 -15593.371} C_VEL
LIN {X 0,Y 311.219,Z 372.089,A -85,B 0,C 180,E1 -15593.433,E2 -15593.433} C_VEL
LIN {X 0,Y 311.56,Z 368.363,A -85,B 0,C 180,E1 -15596.817,E2 -15596.817} C_VEL
LIN {X 0,Y 312.196,Z 363.688,A -85,B 0,C 180,E1 -15601.191,E2 -15601.191} C_VEL
LIN {X 0,Y 312.574,Z 360.615,A -85,B 0,C 180,E1 -15604.201,E2 -15604.201} C_VEL
LIN {X 0,Y 313.034,Z 357.542,A -85,B 0,C 180,E1 -15607.314,E2 -15607.314} C_VEL
LIN {X 0,Y 313.435,Z 354.51,A -85,B 0,C 180,E1 -15610.56,E2 -15610.56} C_VEL
LIN {X 0,Y 313.559,Z 352.953,A -85,B 0,C 180,E1 -15612.298,E2 -15612.298} C_VEL
LIN {X 0,Y 313.559,Z 351.377,A -85,B 0,C 180,E1 -15614.172,E2 -15614.172} C_VEL
LIN {X 0,Y 313.298,Z 348.535,A -85,B 0,C 180,E1 -15617.754,E2 -15617.754} C_VEL
LIN {X 0,Y 312.948,Z 346.181,A -85,B 0,C 180,E1 -15621.037,E2 -15621.037} C_VEL
LIN {X 0,Y 312.668,Z 344.06,A -85,B 0,C 180,E1 -15624.238,E2 -15624.238} C_VEL
LIN {X 0,Y 312.521,Z 343.091,A -85,B 0,C 180,E1 -15625.791,E2 -15625.791} C_VEL
LIN {X 0,Y 312.521,Z 343.057,A -85,B 0,C 180,E1 -15628.853,E2 -15628.853} C_VEL
LIN {X 0,Y 312.571,Z 343.052,A -85,B 0,C 180,E1 -15631.824,E2 -15631.824} C_VEL
LIN {X 0,Y 312.585,Z 343.046,A -85,B 0,C 180,E1 -15634.71,E2 -15634.71} C_VEL
LIN {X 0,Y 312.565,Z 343.053,A -85,B 0,C 180,E1 -15637.527,E2 -15637.527} C_VEL
LIN {X 0,Y 312.582,Z 343.051,A -85,B 0,C 180,E1 -15641.652,E2 -15641.652} C_VEL
LIN {X 0,Y 312.685,Z 343.037,A -85,B 0,C 180,E1 -15645.685,E2 -15645.685} C_VEL
LIN {X 0,Y 312.701,Z 343.034,A -85,B 0,C 180,E1 -15649.641,E2 -15649.641} C_VEL
LIN {X 0,Y 312.866,Z 343.011,A -85,B 0,C 180,E1 -15652.253,E2 -15652.253} C_VEL
LIN {X 0,Y 312.715,Z 343.031,A -85,B 0,C 180,E1 -15654.842,E2 -15654.842} C_VEL
LIN {X 0,Y 312.99,Z 342.995,A -85,B 0,C 180,E1 -15658.713,E2 -15658.713} C_VEL
LIN {X 0,Y 312.988,Z 342.99,A -85,B 0,C 180,E1 -15661.286,E2 -15661.286} C_VEL
LIN {X 0,Y 312.715,Z 343.033,A -85,B 0,C 180,E1 -15665.157,E2 -15665.157} C_VEL
LIN {X 0,Y 312.865,Z 343.011,A -85,B 0,C 180,E1 -15667.745,E2 -15667.745} C_VEL
LIN {X 0,Y 312.668,Z 343.035,A -85,B 0,C 180,E1 -15671.671,E2 -15671.671} C_VEL
LIN {X 0,Y 312.698,Z 343.034,A -85,B 0,C 180,E1 -15674.887,E2 -15674.887} C_VEL
LIN {X 0,Y 312.627,Z 343.039,A -85,B 0,C 180,E1 -15679.235,E2 -15679.235} C_VEL
LIN {X 0,Y 312.524,Z 343.057,A -85,B 0,C 180,E1 -15682.78,E2 -15682.78} C_VEL
LIN {X 0,Y 312.58,Z 343.05,A -85,B 0,C 180,E1 -15686.722,E2 -15686.722} C_VEL
LIN {X 0,Y 312.543,Z 343.051,A -85,B 0,C 180,E1 -15689.649,E2 -15689.649} C_VEL
LIN {X 0,Y 312.517,Z 343.054,A -85,B 0,C 180,E1 -15693.688,E2 -15693.688} C_VEL
LIN {X 0,Y 312.549,Z 343.05,A -85,B 0,C 180,E1 -15697.381,E2 -15697.381} C_VEL
LIN {X 0,Y 312.53,Z 343.054,A -85,B 0,C 180,E1 -15700.702,E2 -15700.702} C_VEL
LIN {X 0,Y 312.536,Z 343.056,A -85,B 0,C 180,E1 -15704.193,E2 -15704.193} C_VEL
LIN {X 0,Y 312.53,Z 343.056,A -85,B 0,C 180,E1 -15707.908,E2 -15707.908} C_VEL
LIN {X 0,Y 312.553,Z 343.055,A -85,B 0,C 180,E1 -15711.905,E2 -15711.905} C_VEL
LIN {X 0,Y 312.503,Z 343.061,A -85,B 0,C 180,E1 -15715.79,E2 -15715.79} C_VEL
LIN {X 0,Y 312.52,Z 343.054,A -85,B 0,C 180,E1 -15718.854,E2 -15718.854} C_VEL
LIN {X 0,Y 312.571,Z 343.052,A -85,B 0,C 180,E1 -15721.825,E2 -15721.825} C_VEL
LIN {X 0,Y 312.582,Z 343.047,A -85,B 0,C 180,E1 -15724.711,E2 -15724.711} C_VEL
LIN {X 0,Y 312.524,Z 343.055,A -85,B 0,C 180,E1 -15726.355,E2 -15726.355} C_VEL
LIN {X 0,Y 313.585,Z 345.974,A -85,B 0,C 180,E1 -15726.529,E2 -15726.529} C_VEL
LIN {X 0,Y 316.617,Z 350.925,A -85,B 0,C 180,E1 -15726.949,E2 -15726.949} C_VEL
LIN {X 0,Y 319.708,Z 355.503,A -85,B 0,C 180,E1 -15727.407,E2 -15727.407} C_VEL
LIN {X 0,Y 323.311,Z 360.404,A -85,B 0,C 180,E1 -15727.997,E2 -15727.997} C_VEL
LIN {X 0,Y 328.112,Z 366.372,A -85,B 0,C 180,E1 -15728.843,E2 -15728.843} C_VEL
LIN {X 0,Y 332.775,Z 371.906,A -85,B 0,C 180,E1 -15729.734,E2 -15729.734} C_VEL
LIN {X 0,Y 337.964,Z 377.845,A -85,B 0,C 180,E1 -15730.818,E2 -15730.818} C_VEL
LIN {X 0,Y 343.83,Z 384.11,A -85,B 0,C 180,E1 -15732.145,E2 -15732.145} C_VEL
LIN {X 0,Y 349.864,Z 390.314,A -85,B 0,C 180,E1 -15733.667,E2 -15733.667} C_VEL
LIN {X 0,Y 352.529,Z 392.494,A -85,B 0,C 180,E1 -15734.345,E2 -15734.345} C_VEL
LIN {X 0,Y 356.93,Z 397.142,A -85,B 0,C 180,E1 -15735.674,E2 -15735.674} C_VEL
LIN {X 0,Y 361.426,Z 401.01,A -85,B 0,C 180,E1 -15737.111,E2 -15737.111} C_VEL
LIN {X 0,Y 365.573,Z 404.856,A -85,B 0,C 180,E1 -15738.65,E2 -15738.65} C_VEL
LIN {X 0,Y 369.375,Z 407.442,A -85,B 0,C 180,E1 -15740.14,E2 -15740.14} C_VEL
LIN {X 0,Y 371.588,Z 409.787,A -85,B 0,C 180,E1 -15741.297,E2 -15741.297} C_VEL
LIN {X 0,Y 373.499,Z 411.695,A -85,B 0,C 180,E1 -15742.431,E2 -15742.431} C_VEL
LIN {X 0,Y 375.251,Z 413.136,A -85,B 0,C 180,E1 -15743.548,E2 -15743.548} C_VEL
LIN {X 0,Y 376.76,Z 414.148,A -85,B 0,C 180,E1 -15744.648,E2 -15744.648} C_VEL
LIN {X 0,Y 378.091,Z 414.725,A -85,B 0,C 180,E1 -15745.736,E2 -15745.736} C_VEL
LIN {X 0,Y 379.826,Z 415.177,A -85,B 0,C 180,E1 -15747.653,E2 -15747.653} C_VEL
LIN {X 0,Y 380.476,Z 415.274,A -85,B 0,C 180,E1 -15748.942,E2 -15748.942} C_VEL
LIN {X 0,Y 380.634,Z 415.322,A -85,B 0,C 180,E1 -15750,E2 -15750} C_VEL
LIN {X 0,Y 380.474,Z 415.277,A -85,B 0,C 180,E1 -15751.058,E2 -15751.058} C_VEL
LIN {X 0,Y 379.822,Z 415.2,A -85,B 0,C 180,E1 -15752.332,E2 -15752.332} C_VEL
LIN {X 0,Y 378.084,Z 414.754,A -85,B 0,C 180,E1 -15754.264,E2 -15754.264} C_VEL
LIN {X 0,Y 376.794,Z 414.122,A -85,B 0,C 180,E1 -15755.351,E2 -15755.351} C_VEL
LIN {X 0,Y 374.979,Z 412.95,A -85,B 0,C 180,E1 -15756.62,E2 -15756.62} C_VEL
LIN {X 0,Y 373.505,Z 411.728,A -85,B 0,C 180,E1 -15757.569,E2 -15757.569} C_VEL
LIN {X 0,Y 370.382,Z 408.467,A -85,B 0,C 180,E1 -15759.36,E2 -15759.36} C_VEL
LIN {X 0,Y 369.38,Z 407.467,A -85,B 0,C 180,E1 -15759.86,E2 -15759.86} C_VEL
LIN {X 0,Y 365.563,Z 404.889,A -85,B 0,C 180,E1 -15761.343,E2 -15761.343} C_VEL
LIN {X 0,Y 361.932,Z 401.561,A -85,B 0,C 180,E1 -15762.697,E2 -15762.697} C_VEL
LIN {X 0,Y 358.274,Z 398.258,A -85,B 0,C 180,E1 -15763.908,E2 -15763.908} C_VEL
LIN {X 0,Y 354.954,Z 395.241,A -85,B 0,C 180,E1 -15764.916,E2 -15764.916} C_VEL
LIN {X 0,Y 351.006,Z 391.252,A -85,B 0,C 180,E1 -15766.041,E2 -15766.041} C_VEL
LIN {X 0,Y 346.967,Z 387.388,A -85,B 0,C 180,E1 -15767.079,E2 -15767.079} C_VEL
LIN {X 0,Y 340.019,Z 380.098,A -85,B 0,C 180,E1 -15768.728,E2 -15768.728} C_VEL
LIN {X 0,Y 333.939,Z 373.269,A -85,B 0,C 180,E1 -15770.031,E2 -15770.031} C_VEL
LIN {X 0,Y 328.852,Z 367.334,A -85,B 0,C 180,E1 -15771.013,E2 -15771.013} C_VEL
LIN {X 0,Y 324.197,Z 361.49,A -85,B 0,C 180,E1 -15771.854,E2 -15771.854} C_VEL
LIN {X 0,Y 320.428,Z 356.558,A -85,B 0,C 180,E1 -15772.477,E2 -15772.477} C_VEL
LIN {X 0,Y 316.877,Z 351.313,A -85,B 0,C 180,E1 -15773.014,E2 -15773.014} C_VEL
LIN {X 0,Y 314.588,Z 347.67,A -85,B 0,C 180,E1 -15773.339,E2 -15773.339} C_VEL
LIN {X 0,Y 312.734,Z 344.09,A -85,B 0,C 180,E1 -15773.595,E2 -15773.595} C_VEL
LIN {X 0,Y 312.535,Z 343.054,A -85,B 0,C 180,E1 -15773.667,E2 -15773.667} C_VEL
LIN {X 0,Y 312.551,Z 343.053,A -85,B 0,C 180,E1 -15776.726,E2 -15776.726} C_VEL
LIN {X 0,Y 312.541,Z 343.052,A -85,B 0,C 180,E1 -15779.65,E2 -15779.65} C_VEL
LIN {X 0,Y 312.516,Z 343.056,A -85,B 0,C 180,E1 -15783.689,E2 -15783.689} C_VEL
LIN {X 0,Y 312.548,Z 343.051,A -85,B 0,C 180,E1 -15787.382,E2 -15787.382} C_VEL
LIN {X 0,Y 312.498,Z 343.057,A -85,B 0,C 180,E1 -15790.708,E2 -15790.708} C_VEL
LIN {X 0,Y 312.529,Z 343.055,A -85,B 0,C 180,E1 -15794.196,E2 -15794.196} C_VEL
LIN {X 0,Y 312.547,Z 343.055,A -85,B 0,C 180,E1 -15797.906,E2 -15797.906} C_VEL
LIN {X 0,Y 312.555,Z 343.053,A -85,B 0,C 180,E1 -15801.905,E2 -15801.905} C_VEL
LIN {X 0,Y 312.503,Z 343.059,A -85,B 0,C 180,E1 -15805.791,E2 -15805.791} C_VEL
LIN {X 0,Y 312.521,Z 343.054,A -85,B 0,C 180,E1 -15808.855,E2 -15808.855} C_VEL
LIN {X 0,Y 312.572,Z 343.05,A -85,B 0,C 180,E1 -15811.825,E2 -15811.825} C_VEL
LIN {X 0,Y 312.582,Z 343.045,A -85,B 0,C 180,E1 -15814.712,E2 -15814.712} C_VEL
LIN {X 0,Y 312.536,Z 343.053,A -85,B 0,C 180,E1 -15818.913,E2 -15818.913} C_VEL
LIN {X 0,Y 312.636,Z 343.041,A -85,B 0,C 180,E1 -15821.657,E2 -15821.657} C_VEL
LIN {X 0,Y 312.692,Z 343.032,A -85,B 0,C 180,E1 -15825.687,E2 -15825.687} C_VEL
LIN {X 0,Y 312.7,Z 343.03,A -85,B 0,C 180,E1 -15829.643,E2 -15829.643} C_VEL
LIN {X 0,Y 312.865,Z 343.011,A -85,B 0,C 180,E1 -15832.255,E2 -15832.255} C_VEL
LIN {X 0,Y 312.715,Z 343.033,A -85,B 0,C 180,E1 -15834.843,E2 -15834.843} C_VEL
LIN {X 0,Y 312.717,Z 343.025,A -85,B 0,C 180,E1 -15836.313,E2 -15836.313} C_VEL
LIN {X 0,Y 312.186,Z 343.089,A -85,B 0,C 180,E1 -15837.392,E2 -15837.392} C_VEL
LIN {X 0,Y 309.456,Z 343.433,A -85,B 0,C 180,E1 -15839.149,E2 -15839.149} C_VEL
LIN {X 0,Y 307.054,Z 343.733,A -85,B 0,C 180,E1 -15840.575,E2 -15840.575} C_VEL
LIN {X 0,Y 305.994,Z 343.866,A -85,B 0,C 180,E1 -15841.677,E2 -15841.677} C_VEL
LIN {X 0,Y 305.897,Z 343.878,A -85,B 0,C 180,E1 -15842.05,E2 -15842.05} C_VEL
LIN {X 0,Y 305.846,Z 343.89,A -85,B 0,C 180,E1 -15846.598,E2 -15846.598} C_VEL
LIN {X 0,Y 305.736,Z 343.9,A -85,B 0,C 180,E1 -15849.26,E2 -15849.26} C_VEL
LIN {X 0,Y 305.587,Z 343.918,A -85,B 0,C 180,E1 -15853.297,E2 -15853.297} C_VEL
LIN {X 0,Y 305.551,Z 343.924,A -85,B 0,C 180,E1 -15856.023,E2 -15856.023} C_VEL
LIN {X 0,Y 305.542,Z 343.923,A -85,B 0,C 180,E1 -15859.427,E2 -15859.427} C_VEL
LIN {X 0,Y 305.487,Z 343.931,A -85,B 0,C 180,E1 -15863.04,E2 -15863.04} C_VEL
LIN {X 0,Y 305.548,Z 343.927,A -85,B 0,C 180,E1 -15866.227,E2 -15866.227} C_VEL
LIN {X 0,Y 305.489,Z 343.931,A -85,B 0,C 180,E1 -15869.048,E2 -15869.048} C_VEL
LIN {X 0,Y 305.469,Z 343.939,A -85,B 0,C 180,E1 -15873.517,E2 -15873.517} C_VEL
LIN {X 0,Y 305.706,Z 345.76,A -85,B 0,C 180,E1 -15876.708,E2 -15876.708} C_VEL
LIN {X 0,Y 306.13,Z 348.477,A -85,B 0,C 180,E1 -15880.747,E2 -15880.747} C_VEL
LIN {X 0,Y 306.371,Z 350.506,A -85,B 0,C 180,E1 -15883.488,E2 -15883.488} C_VEL
LIN {X 0,Y 306.512,Z 352.939,A -85,B 0,C 180,E1 -15886.539,E2 -15886.539} C_VEL
LIN {X 0,Y 306.318,Z 355.941,A -85,B 0,C 180,E1 -15890.028,E2 -15890.028} C_VEL
LIN {X 0,Y 305.856,Z 359.177,A -85,B 0,C 180,E1 -15893.537,E2 -15893.537} C_VEL
LIN {X 0,Y 305.4,Z 362.029,A -85,B 0,C 180,E1 -15896.475,E2 -15896.475} C_VEL
LIN {X 0,Y 304.97,Z 365.107,A -85,B 0,C 180,E1 -15899.537,E2 -15899.537} C_VEL
LIN {X 0,Y 304.373,Z 370.032,A -85,B 0,C 180,E1 -15904.227,E2 -15904.227} C_VEL
LIN {X 0,Y 304.199,Z 371.932,A -85,B 0,C 180,E1 -15906.005,E2 -15906.005} C_VEL
LIN {X 0,Y 307.819,Z 386.736,A -85,B 0,C 180,E1 -15907.006,E2 -15907.006} C_VEL
LIN {X 0,Y 309.985,Z 398.779,A -85,B 0,C 180,E1 -15908.035,E2 -15908.035} C_VEL
LIN {X 0,Y 311.203,Z 408.334,A -85,B 0,C 180,E1 -15908.991,E2 -15908.991} C_VEL
LIN {X 0,Y 311.802,Z 416.306,A -85,B 0,C 180,E1 -15909.896,E2 -15909.896} C_VEL
LIN {X 0,Y 310.348,Z 426.602,A -85,B 0,C 180,E1 -15911.174,E2 -15911.174} C_VEL
LIN {X 0,Y 309.03,Z 435.131,A -85,B 0,C 180,E1 -15912.462,E2 -15912.462} C_VEL
LIN {X 0,Y 308.02,Z 442.334,A -85,B 0,C 180,E1 -15913.765,E2 -15913.765} C_VEL
LIN {X 0,Y 307.087,Z 448.557,A -85,B 0,C 180,E1 -15915.08,E2 -15915.08} C_VEL
LIN {X 0,Y 305.958,Z 455.093,A -85,B 0,C 180,E1 -15916.72,E2 -15916.72} C_VEL
LIN {X 0,Y 305.223,Z 459.594,A -85,B 0,C 180,E1 -15918.04,E2 -15918.04} C_VEL
LIN {X 0,Y 304.482,Z 465.088,A -85,B 0,C 180,E1 -15920.031,E2 -15920.031} C_VEL
LIN {X 0,Y 303.993,Z 469.416,A -85,B 0,C 180,E1 -15922.027,E2 -15922.027} C_VEL
LIN {X 0,Y 303.751,Z 471.783,A -85,B 0,C 180,E1 -15923.357,E2 -15923.357} C_VEL
LIN {X 0,Y 303.64,Z 473.585,A -85,B 0,C 180,E1 -15924.688,E2 -15924.688} C_VEL
LIN {X 0,Y 303.608,Z 476.035,A -85,B 0,C 180,E1 -15927.346,E2 -15927.346} C_VEL
LIN {X 0,Y 303.567,Z 476.624,A -85,B 0,C 180,E1 -15928.673,E2 -15928.673} C_VEL
LIN {X 0,Y 303.567,Z 476.624,A -85,B 0,C 180,E1 -15931.327,E2 -15931.327} C_VEL
LIN {X 0,Y 303.608,Z 476.035,A -85,B 0,C 180,E1 -15932.654,E2 -15932.654} C_VEL
LIN {X 0,Y 303.64,Z 473.584,A -85,B 0,C 180,E1 -15935.312,E2 -15935.312} C_VEL
LIN {X 0,Y 303.844,Z 470.633,A -85,B 0,C 180,E1 -15937.309,E2 -15937.309} C_VEL
LIN {X 0,Y 304.304,Z 466.643,A -85,B 0,C 180,E1 -15939.304,E2 -15939.304} C_VEL
LIN {X 0,Y 304.979,Z 461.512,A -85,B 0,C 180,E1 -15941.296,E2 -15941.296} C_VEL
LIN {X 0,Y 305.752,Z 456.248,A -85,B 0,C 180,E1 -15942.951,E2 -15942.951} C_VEL
LIN {X 0,Y 306.838,Z 449.933,A -85,B 0,C 180,E1 -15944.593,E2 -15944.593} C_VEL
LIN {X 0,Y 307.751,Z 443.98,A -85,B 0,C 180,E1 -15945.905,E2 -15945.905} C_VEL
LIN {X 0,Y 308.746,Z 437.05,A -85,B 0,C 180,E1 -15947.213,E2 -15947.213} C_VEL
LIN {X 0,Y 309.808,Z 430.005,A -85,B 0,C 180,E1 -15948.346,E2 -15948.346} C_VEL
LIN {X 0,Y 311.073,Z 421.713,A -85,B 0,C 180,E1 -15949.466,E2 -15949.466} C_VEL
LIN {X 0,Y 311.79,Z 416.305,A -85,B 0,C 180,E1 -15950.105,E2 -15950.105} C_VEL
LIN {X 0,Y 310.798,Z 404.948,A -85,B 0,C 180,E1 -15951.375,E2 -15951.375} C_VEL
LIN {X 0,Y 309.252,Z 393.967,A -85,B 0,C 180,E1 -15952.392,E2 -15952.392} C_VEL
LIN {X 0,Y 306.955,Z 382.932,A -85,B 0,C 180,E1 -15953.262,E2 -15953.262} C_VEL
LIN {X 0,Y 304.24,Z 372.574,A -85,B 0,C 180,E1 -15953.948,E2 -15953.948} C_VEL
LIN {X 0,Y 304.177,Z 371.928,A -85,B 0,C 180,E1 -15954,E2 -15954} C_VEL
LIN {X 0,Y 304.546,Z 368.194,A -85,B 0,C 180,E1 -15957.486,E2 -15957.486} C_VEL
LIN {X 0,Y 305.166,Z 363.985,A -85,B 0,C 180,E1 -15961.557,E2 -15961.557} C_VEL
LIN {X 0,Y 305.615,Z 360.484,A -85,B 0,C 180,E1 -15965.093,E2 -15965.093} C_VEL
LIN {X 0,Y 306.157,Z 357.07,A -85,B 0,C 180,E1 -15968.694,E2 -15968.694} C_VEL
LIN {X 0,Y 306.453,Z 354.412,A -85,B 0,C 180,E1 -15971.687,E2 -15971.687} C_VEL
LIN {X 0,Y 306.46,Z 351.429,A -85,B 0,C 180,E1 -15975.309,E2 -15975.309} C_VEL
LIN {X 0,Y 306.132,Z 348.475,A -85,B 0,C 180,E1 -15979.252,E2 -15979.252} C_VEL
LIN {X 0,Y 305.705,Z 345.764,A -85,B 0,C 180,E1 -15983.292,E2 -15983.292} C_VEL
LIN {X 0,Y 305.469,Z 343.94,A -85,B 0,C 180,E1 -15986.483,E2 -15986.483} C_VEL
LIN {X 0,Y 305.489,Z 343.931,A -85,B 0,C 180,E1 -15990.952,E2 -15990.952} C_VEL
LIN {X 0,Y 305.572,Z 343.923,A -85,B 0,C 180,E1 -15994.087,E2 -15994.087} C_VEL
LIN {X 0,Y 305.476,Z 343.933,A -85,B 0,C 180,E1 -15998.4,E2 -15998.4} C_VEL
LIN {X 0,Y 305.543,Z 343.925,A -85,B 0,C 180,E1 -16001.214,E2 -16001.214} C_VEL
LIN {X 0,Y 305.626,Z 343.916,A -85,B 0,C 180,E1 -16005.347,E2 -16005.347} C_VEL
LIN {X 0,Y 305.639,Z 343.916,A -85,B 0,C 180,E1 -16009.399,E2 -16009.399} C_VEL
LIN {X 0,Y 305.808,Z 343.89,A -85,B 0,C 180,E1 -16012.073,E2 -16012.073} C_VEL
LIN {X 0,Y 305.686,Z 343.906,A -85,B 0,C 180,E1 -16014.723,E2 -16014.723} C_VEL
LIN {X 0,Y 305.957,Z 343.871,A -85,B 0,C 180,E1 -16018.683,E2 -16018.683} C_VEL
LIN {X 0,Y 305.955,Z 343.865,A -85,B 0,C 180,E1 -16021.316,E2 -16021.316} C_VEL
LIN {X 0,Y 305.686,Z 343.908,A -85,B 0,C 180,E1 -16025.276,E2 -16025.276} C_VEL
LIN {X 0,Y 305.807,Z 343.889,A -85,B 0,C 180,E1 -16027.925,E2 -16027.925} C_VEL
LIN {X 0,Y 305.602,Z 343.915,A -85,B 0,C 180,E1 -16031.944,E2 -16031.944} C_VEL
LIN {X 0,Y 305.636,Z 343.914,A -85,B 0,C 180,E1 -16035.034,E2 -16035.034} C_VEL
LIN {X 0,Y 305.574,Z 343.917,A -85,B 0,C 180,E1 -16039.444,E2 -16039.444} C_VEL
LIN {X 0,Y 305.484,Z 343.931,A -85,B 0,C 180,E1 -16043.039,E2 -16043.039} C_VEL
LIN {X 0,Y 305.551,Z 343.923,A -85,B 0,C 180,E1 -16046.229,E2 -16046.229} C_VEL
LIN {X 0,Y 305.493,Z 343.93,A -85,B 0,C 180,E1 -16049.049,E2 -16049.049} C_VEL
LIN {X 0,Y 305.442,Z 343.937,A -85,B 0,C 180,E1 -16051.951,E2 -16051.951} C_VEL
LIN {X 0,Y 305.46,Z 343.933,A -85,B 0,C 180,E1 -16055.113,E2 -16055.113} C_VEL
LIN {X 0,Y 305.491,Z 343.932,A -85,B 0,C 180,E1 -16058.539,E2 -16058.539} C_VEL
LIN {X 0,Y 305.507,Z 343.929,A -85,B 0,C 180,E1 -16062.597,E2 -16062.597} C_VEL
LIN {X 0,Y 305.485,Z 343.932,A -85,B 0,C 180,E1 -16066.356,E2 -16066.356} C_VEL
LIN {X 0,Y 305.462,Z 343.937,A -85,B 0,C 180,E1 -16069.893,E2 -16069.893} C_VEL
LIN {X 0,Y 305.498,Z 343.932,A -85,B 0,C 180,E1 -16073.626,E2 -16073.626} C_VEL
LIN {X 0,Y 305.461,Z 343.934,A -85,B 0,C 180,E1 -16076.483,E2 -16076.483} C_VEL
LIN {X 0,Y 305.46,Z 343.937,A -85,B 0,C 180,E1 -16079.591,E2 -16079.591} C_VEL
LIN {X 0,Y 305.517,Z 343.927,A -85,B 0,C 180,E1 -16082.608,E2 -16082.608} C_VEL
LIN {X 0,Y 305.498,Z 343.933,A -85,B 0,C 180,E1 -16085.749,E2 -16085.749} C_VEL
LIN {X 0,Y 306.513,Z 346.813,A -85,B 0,C 180,E1 -16085.927,E2 -16085.927} C_VEL
LIN {X 0,Y 310.955,Z 354.769,A -85,B 0,C 180,E1 -16086.52,E2 -16086.52} C_VEL
LIN {X 0,Y 316.664,Z 363.085,A -85,B 0,C 180,E1 -16087.385,E2 -16087.385} C_VEL
LIN {X 0,Y 323.41,Z 371.415,A -85,B 0,C 180,E1 -16088.535,E2 -16088.535} C_VEL
LIN {X 0,Y 329.626,Z 378.788,A -85,B 0,C 180,E1 -16089.737,E2 -16089.737} C_VEL
LIN {X 0,Y 336.705,Z 386.743,A -85,B 0,C 180,E1 -16091.278,E2 -16091.278} C_VEL
LIN {X 0,Y 342.752,Z 392.949,A -85,B 0,C 180,E1 -16092.714,E2 -16092.714} C_VEL
LIN {X 0,Y 346.845,Z 396.921,A -85,B 0,C 180,E1 -16093.773,E2 -16093.773} C_VEL
LIN {X 0,Y 349.866,Z 399.851,A -85,B 0,C 180,E1 -16094.622,E2 -16094.622} C_VEL
LIN {X 0,Y 352.762,Z 402.798,A -85,B 0,C 180,E1 -16095.501,E2 -16095.501} C_VEL
LIN {X 0,Y 357.206,Z 406.6,A -85,B 0,C 180,E1 -16096.908,E2 -16096.908} C_VEL
LIN {X 0,Y 361.421,Z 410.581,A -85,B 0,C 180,E1 -16098.469,E2 -16098.469} C_VEL
LIN {X 0,Y 365.471,Z 413.368,A -85,B 0,C 180,E1 -16100.034,E2 -16100.034} C_VEL
LIN {X 0,Y 369.051,Z 417.039,A -85,B 0,C 180,E1 -16101.991,E2 -16101.991} C_VEL
LIN {X 0,Y 371.393,Z 419.062,A -85,B 0,C 180,E1 -16103.481,E2 -16103.481} C_VEL
LIN {X 0,Y 373.76,Z 420.516,A -85,B 0,C 180,E1 -16105.256,E2 -16105.256} C_VEL
LIN {X 0,Y 375.389,Z 421.032,A -85,B 0,C 180,E1 -16106.78,E2 -16106.78} C_VEL
LIN {X 0,Y 376.236,Z 421.208,A -85,B 0,C 180,E1 -16107.859,E2 -16107.859} C_VEL
LIN {X 0,Y 376.75,Z 421.309,A -85,B 0,C 180,E1 -16108.931,E2 -16108.931} C_VEL
LIN {X 0,Y 376.918,Z 421.356,A -85,B 0,C 180,E1 -16110,E2 -16110} C_VEL
LIN {X 0,Y 376.749,Z 421.311,A -85,B 0,C 180,E1 -16111.069,E2 -16111.069} C_VEL
LIN {X 0,Y 376.207,Z 421.244,A -85,B 0,C 180,E1 -16112.141,E2 -16112.141} C_VEL
LIN {X 0,Y 375.39,Z 421.019,A -85,B 0,C 180,E1 -16113.22,E2 -16113.22} C_VEL
LIN {X 0,Y 373.76,Z 420.502,A -85,B 0,C 180,E1 -16114.745,E2 -16114.745} C_VEL
LIN {X 0,Y 371.352,Z 419.087,A -85,B 0,C 180,E1 -16116.52,E2 -16116.52} C_VEL
LIN {X 0,Y 369.05,Z 417.059,A -85,B 0,C 180,E1 -16118.008,E2 -16118.008} C_VEL
LIN {X 0,Y 365.473,Z 413.378,A -85,B 0,C 180,E1 -16119.966,E2 -16119.966} C_VEL
LIN {X 0,Y 361.416,Z 410.569,A -85,B 0,C 180,E1 -16121.533,E2 -16121.533} C_VEL
LIN {X 0,Y 357.187,Z 406.582,A -85,B 0,C 180,E1 -16123.094,E2 -16123.094} C_VEL
LIN {X 0,Y 352.729,Z 402.76,A -85,B 0,C 180,E1 -16124.501,E2 -16124.501} C_VEL
LIN {X 0,Y 346.848,Z 396.917,A -85,B 0,C 180,E1 -16126.232,E2 -16126.232} C_VEL
LIN {X 0,Y 341.835,Z 391.859,A -85,B 0,C 180,E1 -16127.529,E2 -16127.529} C_VEL
LIN {X 0,Y 335.759,Z 385.62,A -85,B 0,C 180,E1 -16128.945,E2 -16128.945} C_VEL
LIN {X 0,Y 329.626,Z 378.766,A -85,B 0,C 180,E1 -16130.263,E2 -16130.263} C_VEL
LIN {X 0,Y 324.176,Z 372.381,A -85,B 0,C 180,E1 -16131.317,E2 -16131.317} C_VEL
LIN {X 0,Y 319.549,Z 366.635,A -85,B 0,C 180,E1 -16132.147,E2 -16132.147} C_VEL
LIN {X 0,Y 315.288,Z 361.023,A -85,B 0,C 180,E1 -16132.844,E2 -16132.844} C_VEL
LIN {X 0,Y 310.113,Z 353.472,A -85,B 0,C 180,E1 -16133.596,E2 -16133.596} C_VEL
LIN {X 0,Y 305.783,Z 345.202,A -85,B 0,C 180,E1 -16134.175,E2 -16134.175} C_VEL
LIN {X 0,Y 305.492,Z 343.934,A -85,B 0,C 180,E1 -16134.268,E2 -16134.268} C_VEL
LIN {X 0,Y 305.517,Z 343.927,A -85,B 0,C 180,E1 -16137.392,E2 -16137.392} C_VEL
LIN {X 0,Y 305.46,Z 343.937,A -85,B 0,C 180,E1 -16140.409,E2 -16140.409} C_VEL
LIN {X 0,Y 305.461,Z 343.938,A -85,B 0,C 180,E1 -16144.079,E2 -16144.079} C_VEL
LIN {X 0,Y 305.498,Z 343.929,A -85,B 0,C 180,E1 -16146.736,E2 -16146.736} C_VEL
LIN {X 0,Y 305.462,Z 343.937,A -85,B 0,C 180,E1 -16150.107,E2 -16150.107} C_VEL
LIN {X 0,Y 305.485,Z 343.932,A -85,B 0,C 180,E1 -16153.644,E2 -16153.644} C_VEL
LIN {X 0,Y 305.507,Z 343.929,A -85,B 0,C 180,E1 -16157.403,E2 -16157.403} C_VEL
LIN {X 0,Y 305.517,Z 343.93,A -85,B 0,C 180,E1 -16161.605,E2 -16161.605} C_VEL
LIN {X 0,Y 305.459,Z 343.933,A -85,B 0,C 180,E1 -16164.887,E2 -16164.887} C_VEL
LIN {X 0,Y 305.45,Z 343.934,A -85,B 0,C 180,E1 -16168.355,E2 -16168.355} C_VEL
LIN {X 0,Y 305.518,Z 343.928,A -85,B 0,C 180,E1 -16171.114,E2 -16171.114} C_VEL
LIN {X 0,Y 305.569,Z 343.919,A -85,B 0,C 180,E1 -16174.089,E2 -16174.089} C_VEL
LIN {X 0,Y 305.48,Z 343.93,A -85,B 0,C 180,E1 -16178.402,E2 -16178.402} C_VEL
LIN {X 0,Y 305.588,Z 343.92,A -85,B 0,C 180,E1 -16181.218,E2 -16181.218} C_VEL
LIN {X 0,Y 305.647,Z 343.912,A -85,B 0,C 180,E1 -16185.35,E2 -16185.35} C_VEL
LIN {X 0,Y 305.637,Z 343.912,A -85,B 0,C 180,E1 -16189.4,E2 -16189.4} C_VEL
LIN {X 0,Y 305.807,Z 343.889,A -85,B 0,C 180,E1 -16192.075,E2 -16192.075} C_VEL
LIN {X 0,Y 305.686,Z 343.908,A -85,B 0,C 180,E1 -16194.724,E2 -16194.724} C_VEL
LIN {X 0,Y 305.955,Z 343.865,A -85,B 0,C 180,E1 -16198.684,E2 -16198.684} C_VEL
LIN {X 0,Y 305.957,Z 343.871,A -85,B 0,C 180,E1 -16201.317,E2 -16201.317} C_VEL
LIN {X 0,Y 305.897,Z 343.878,A -85,B 0,C 180,E1 -16202.05,E2 -16202.05} C_VEL
LIN {X 0,Y 305.19,Z 343.971,A -85,B 0,C 180,E1 -16203.147,E2 -16203.147} C_VEL
LIN {X 0,Y 302.288,Z 344.332,A -85,B 0,C 180,E1 -16204.932,E2 -16204.932} C_VEL
LIN {X 0,Y 299.855,Z 344.634,A -85,B 0,C 180,E1 -16206.381,E2 -16206.381} C_VEL
LIN {X 0,Y 298.826,Z 344.76,A -85,B 0,C 180,E1 -16207.503,E2 -16207.503} C_VEL
LIN {X 0,Y 298.749,Z 344.77,A -85,B 0,C 180,E1 -16207.883,E2 -16207.883} C_VEL
LIN {X 0,Y 298.594,Z 344.792,A -85,B 0,C 180,E1 -16210.854,E2 -16210.854} C_VEL
LIN {X 0,Y 298.548,Z 344.796,A -85,B 0,C 180,E1 -16215.169,E2 -16215.169} C_VEL
LIN {X 0,Y 298.504,Z 344.8,A -85,B 0,C 180,E1 -16219.246,E2 -16219.246} C_VEL
LIN {X 0,Y 298.429,Z 344.811,A -85,B 0,C 180,E1 -16223.601,E2 -16223.601} C_VEL
LIN {X 0,Y 298.49,Z 344.805,A -85,B 0,C 180,E1 -16226.575,E2 -16226.575} C_VEL
LIN {X 0,Y 298.418,Z 344.813,A -85,B 0,C 180,E1 -16229.642,E2 -16229.642} C_VEL
LIN {X 0,Y 298.398,Z 344.819,A -85,B 0,C 180,E1 -16232.801,E2 -16232.801} C_VEL
LIN {X 0,Y 298.53,Z 345.506,A -85,B 0,C 180,E1 -16234.516,E2 -16234.516} C_VEL
LIN {X 0,Y 298.772,Z 347.49,A -85,B 0,C 180,E1 -16237.706,E2 -16237.706} C_VEL
LIN {X 0,Y 299.155,Z 349.864,A -85,B 0,C 180,E1 -16241.256,E2 -16241.256} C_VEL
LIN {X 0,Y 299.476,Z 352.835,A -85,B 0,C 180,E1 -16245.249,E2 -16245.249} C_VEL
LIN {X 0,Y 299.375,Z 355.829,A -85,B 0,C 180,E1 -16248.905,E2 -16248.905} C_VEL
LIN {X 0,Y 298.931,Z 358.847,A -85,B 0,C 180,E1 -16252.319,E2 -16252.319} C_VEL
LIN {X 0,Y 298.469,Z 361.901,A -85,B 0,C 180,E1 -16255.589,E2 -16255.589} C_VEL
LIN {X 0,Y 298.041,Z 364.982,A -85,B 0,C 180,E1 -16258.75,E2 -16258.75} C_VEL
LIN {X 0,Y 297.373,Z 369.596,A -85,B 0,C 180,E1 -16263.318,E2 -16263.318} C_VEL
LIN {X 0,Y 297.167,Z 371.974,A -85,B 0,C 180,E1 -16265.432,E2 -16265.432} C_VEL
LIN {X 0,Y 299.845,Z 382.351,A -85,B 0,C 180,E1 -16266.133,E2 -16266.133} C_VEL
LIN {X 0,Y 302.106,Z 392.795,A -85,B 0,C 180,E1 -16266.981,E2 -16266.981} C_VEL
LIN {X 0,Y 303.545,Z 401.926,A -85,B 0,C 180,E1 -16267.84,E2 -16267.84} C_VEL
LIN {X 0,Y 304.555,Z 411.414,A -85,B 0,C 180,E1 -16268.865,E2 -16268.865} C_VEL
LIN {X 0,Y 304.956,Z 417.462,A -85,B 0,C 180,E1 -16269.6,E2 -16269.6} C_VEL
LIN {X 0,Y 303.636,Z 426.406,A -85,B 0,C 180,E1 -16270.741,E2 -16270.741} C_VEL
LIN {X 0,Y 302.243,Z 434.934,A -85,B 0,C 180,E1 -16272.055,E2 -16272.055} C_VEL
LIN {X 0,Y 301.129,Z 442.449,A -85,B 0,C 180,E1 -16273.45,E2 -16273.45} C_VEL
LIN {X 0,Y 299.927,Z 449.736,A -85,B 0,C 180,E1 -16275.063,E2 -16275.063} C_VEL
LIN {X 0,Y 298.815,Z 456.051,A -85,B 0,C 180,E1 -16276.743,E2 -16276.743} C_VEL
LIN {X 0,Y 297.969,Z 461.314,A -85,B 0,C 180,E1 -16278.435,E2 -16278.435} C_VEL
LIN {X 0,Y 297.27,Z 466.447,A -85,B 0,C 180,E1 -16280.474,E2 -16280.474} C_VEL
LIN {X 0,Y 296.799,Z 470.437,A -85,B 0,C 180,E1 -16282.517,E2 -16282.517} C_VEL
LIN {X 0,Y 296.554,Z 473.388,A -85,B 0,C 180,E1 -16284.56,E2 -16284.56} C_VEL
LIN {X 0,Y 296.535,Z 475.839,A -85,B 0,C 180,E1 -16287.283,E2 -16287.283} C_VEL
LIN {X 0,Y 296.487,Z 476.428,A -85,B 0,C 180,E1 -16288.642,E2 -16288.642} C_VEL
LIN {X 0,Y 296.487,Z 476.428,A -85,B 0,C 180,E1 -16291.358,E2 -16291.358} C_VEL
LIN {X 0,Y 296.534,Z 475.839,A -85,B 0,C 180,E1 -16292.717,E2 -16292.717} C_VEL
LIN {X 0,Y 296.549,Z 473.297,A -85,B 0,C 180,E1 -16295.509,E2 -16295.509} C_VEL
LIN {X 0,Y 296.797,Z 470.437,A -85,B 0,C 180,E1 -16297.483,E2 -16297.483} C_VEL
LIN {X 0,Y 297.27,Z 466.447,A -85,B 0,C 180,E1 -16299.526,E2 -16299.526} C_VEL
LIN {X 0,Y 297.969,Z 461.314,A -85,B 0,C 180,E1 -16301.565,E2 -16301.565} C_VEL
LIN {X 0,Y 298.816,Z 456.051,A -85,B 0,C 180,E1 -16303.257,E2 -16303.257} C_VEL
LIN {X 0,Y 299.933,Z 449.736,A -85,B 0,C 180,E1 -16304.937,E2 -16304.937} C_VEL
LIN {X 0,Y 300.916,Z 443.784,A -85,B 0,C 180,E1 -16306.276,E2 -16306.276} C_VEL
LIN {X 0,Y 301.942,Z 436.854,A -85,B 0,C 180,E1 -16307.613,E2 -16307.613} C_VEL
LIN {X 0,Y 303.223,Z 428.673,A -85,B 0,C 180,E1 -16308.934,E2 -16308.934} C_VEL
LIN {X 0,Y 304.577,Z 420.165,A -85,B 0,C 180,E1 -16310.074,E2 -16310.074} C_VEL
LIN {X 0,Y 304.956,Z 416.104,A -85,B 0,C 180,E1 -16310.576,E2 -16310.576} C_VEL
LIN {X 0,Y 303.734,Z 403.26,A -85,B 0,C 180,E1 -16312.028,E2 -16312.028} C_VEL
LIN {X 0,Y 302.129,Z 392.624,A -85,B 0,C 180,E1 -16313.029,E2 -16313.029} C_VEL
LIN {X 0,Y 299.853,Z 382.277,A -85,B 0,C 180,E1 -16313.87,E2 -16313.87} C_VEL
LIN {X 0,Y 297.219,Z 372.443,A -85,B 0,C 180,E1 -16314.548,E2 -16314.548} C_VEL
LIN {X 0,Y 297.153,Z 371.758,A -85,B 0,C 180,E1 -16314.602,E2 -16314.602} C_VEL
LIN {X 0,Y 297.569,Z 368.044,A -85,B 0,C 180,E1 -16318.187,E2 -16318.187} C_VEL
LIN {X 0,Y 298.127,Z 364.276,A -85,B 0,C 180,E1 -16321.933,E2 -16321.933} C_VEL
LIN {X 0,Y 298.691,Z 360.353,A -85,B 0,C 180,E1 -16326.031,E2 -16326.031} C_VEL
LIN {X 0,Y 299.176,Z 357.304,A -85,B 0,C 180,E1 -16329.365,E2 -16329.365} C_VEL
LIN {X 0,Y 299.473,Z 354.312,A -85,B 0,C 180,E1 -16332.888,E2 -16332.888} C_VEL
LIN {X 0,Y 299.44,Z 352.437,A -85,B 0,C 180,E1 -16335.241,E2 -16335.241} C_VEL
LIN {X 0,Y 299.133,Z 349.779,A -85,B 0,C 180,E1 -16338.863,E2 -16338.863} C_VEL
LIN {X 0,Y 298.771,Z 347.465,A -85,B 0,C 180,E1 -16342.294,E2 -16342.294} C_VEL
LIN {X 0,Y 298.508,Z 345.447,A -85,B 0,C 180,E1 -16345.593,E2 -16345.593} C_VEL
LIN {X 0,Y 298.398,Z 344.821,A -85,B 0,C 180,E1 -16347.199,E2 -16347.199} C_VEL
LIN {X 0,Y 298.428,Z 344.812,A -85,B 0,C 180,E1 -16350.616,E2 -16350.616} C_VEL
LIN {X 0,Y 298.484,Z 344.805,A -85,B 0,C 180,E1 -16353.474,E2 -16353.474} C_VEL
LIN {X 0,Y 298.431,Z 344.81,A -85,B 0,C 180,E1 -16356.699,E2 -16356.699} C_VEL
LIN {X 0,Y 298.504,Z 344.801,A -85,B 0,C 180,E1 -16360.754,E2 -16360.754} C_VEL
LIN {X 0,Y 298.586,Z 344.791,A -85,B 0,C 180,E1 -16364.994,E2 -16364.994} C_VEL
LIN {X 0,Y 298.594,Z 344.791,A -85,B 0,C 180,E1 -16369.146,E2 -16369.146} C_VEL
LIN {X 0,Y 298.755,Z 344.77,A -85,B 0,C 180,E1 -16371.885,E2 -16371.885} C_VEL
LIN {X 0,Y 298.657,Z 344.781,A -85,B 0,C 180,E1 -16374.598,E2 -16374.598} C_VEL
LIN {X 0,Y 298.923,Z 344.747,A -85,B 0,C 180,E1 -16378.652,E2 -16378.652} C_VEL
LIN {X 0,Y 298.922,Z 344.739,A -85,B 0,C 180,E1 -16381.346,E2 -16381.346} C_VEL
LIN {X 0,Y 298.791,Z 344.766,A -85,B 0,C 180,E1 -16386.753,E2 -16386.753} C_VEL
LIN {X 0,Y 298.679,Z 344.777,A -85,B 0,C 180,E1 -16389.48,E2 -16389.48} C_VEL
LIN {X 0,Y 298.551,Z 344.793,A -85,B 0,C 180,E1 -16393.615,E2 -16393.615} C_VEL
LIN {X 0,Y 298.547,Z 344.795,A -85,B 0,C 180,E1 -16396.408,E2 -16396.408} C_VEL
LIN {X 0,Y 298.508,Z 344.796,A -85,B 0,C 180,E1 -16399.653,E2 -16399.653} C_VEL
LIN {X 0,Y 298.426,Z 344.809,A -85,B 0,C 180,E1 -16403.599,E2 -16403.599} C_VEL
LIN {X 0,Y 298.489,Z 344.806,A -85,B 0,C 180,E1 -16406.574,E2 -16406.574} C_VEL
LIN {X 0,Y 298.418,Z 344.811,A -85,B 0,C 180,E1 -16409.64,E2 -16409.64} C_VEL
LIN {X 0,Y 298.393,Z 344.815,A -85,B 0,C 180,E1 -16412.799,E2 -16412.799} C_VEL
LIN {X 0,Y 298.467,Z 344.806,A -85,B 0,C 180,E1 -16416.813,E2 -16416.813} C_VEL
LIN {X 0,Y 298.452,Z 344.806,A -85,B 0,C 180,E1 -16421.102,E2 -16421.102} C_VEL
LIN {X 0,Y 298.415,Z 344.81,A -85,B 0,C 180,E1 -16424.952,E2 -16424.952} C_VEL
LIN {X 0,Y 298.433,Z 344.808,A -85,B 0,C 180,E1 -16426.926,E2 -16426.926} C_VEL
LIN {X 0,Y 298.428,Z 344.809,A -85,B 0,C 180,E1 -16430.999,E2 -16430.999} C_VEL
LIN {X 0,Y 298.43,Z 344.813,A -85,B 0,C 180,E1 -16433.932,E2 -16433.932} C_VEL
LIN {X 0,Y 298.392,Z 344.818,A -85,B 0,C 180,E1 -16437.983,E2 -16437.983} C_VEL
LIN {X 0,Y 298.46,Z 344.809,A -85,B 0,C 180,E1 -16441.904,E2 -16441.904} C_VEL
LIN {X 0,Y 298.48,Z 344.827,A -85,B 0,C 180,E1 -16445.179,E2 -16445.179} C_VEL
LIN {X 0,Y 299.487,Z 347.669,A -85,B 0,C 180,E1 -16445.342,E2 -16445.342} C_VEL
LIN {X 0,Y 303.191,Z 354.991,A -85,B 0,C 180,E1 -16445.875,E2 -16445.875} C_VEL
LIN {X 0,Y 307.843,Z 362.604,A -85,B 0,C 180,E1 -16446.557,E2 -16446.557} C_VEL
LIN {X 0,Y 313.739,Z 370.53,A -85,B 0,C 180,E1 -16447.489,E2 -16447.489} C_VEL
LIN {X 0,Y 320.291,Z 378.697,A -85,B 0,C 180,E1 -16448.66,E2 -16448.66} C_VEL
LIN {X 0,Y 327.128,Z 386.631,A -85,B 0,C 180,E1 -16450.036,E2 -16450.036} C_VEL
LIN {X 0,Y 332.056,Z 392.01,A -85,B 0,C 180,E1 -16451.118,E2 -16451.118} C_VEL
LIN {X 0,Y 338.622,Z 398.802,A -85,B 0,C 180,E1 -16452.689,E2 -16452.689} C_VEL
LIN {X 0,Y 345.04,Z 404.923,A -85,B 0,C 180,E1 -16454.401,E2 -16454.401} C_VEL
LIN {X 0,Y 348.492,Z 408.449,A -85,B 0,C 180,E1 -16455.465,E2 -16455.465} C_VEL
LIN {X 0,Y 351.941,Z 411.323,A -85,B 0,C 180,E1 -16456.523,E2 -16456.523} C_VEL
LIN {X 0,Y 355.883,Z 415.157,A -85,B 0,C 180,E1 -16457.964,E2 -16457.964} C_VEL
LIN {X 0,Y 358.174,Z 417.048,A -85,B 0,C 180,E1 -16458.835,E2 -16458.835} C_VEL
LIN {X 0,Y 360.983,Z 418.911,A -85,B 0,C 180,E1 -16459.909,E2 -16459.909} C_VEL
LIN {X 0,Y 363.278,Z 421.172,A -85,B 0,C 180,E1 -16461.097,E2 -16461.097} C_VEL
LIN {X 0,Y 365.223,Z 423.134,A -85,B 0,C 180,E1 -16462.259,E2 -16462.259} C_VEL
LIN {X 0,Y 367.583,Z 425.038,A -85,B 0,C 180,E1 -16463.827,E2 -16463.827} C_VEL
LIN {X 0,Y 369.921,Z 426.354,A -85,B 0,C 180,E1 -16465.642,E2 -16465.642} C_VEL
LIN {X 0,Y 371.127,Z 426.714,A -85,B 0,C 180,E1 -16466.743,E2 -16466.743} C_VEL
LIN {X 0,Y 372.015,Z 426.932,A -85,B 0,C 180,E1 -16467.835,E2 -16467.835} C_VEL
LIN {X 0,Y 372.573,Z 427.036,A -85,B 0,C 180,E1 -16468.919,E2 -16468.919} C_VEL
LIN {X 0,Y 372.753,Z 427.082,A -85,B 0,C 180,E1 -16470,E2 -16470} C_VEL
LIN {X 0,Y 372.549,Z 427.046,A -85,B 0,C 180,E1 -16471.108,E2 -16471.108} C_VEL
LIN {X 0,Y 371.988,Z 426.959,A -85,B 0,C 180,E1 -16472.165,E2 -16472.165} C_VEL
LIN {X 0,Y 371.124,Z 426.707,A -85,B 0,C 180,E1 -16473.257,E2 -16473.257} C_VEL
LIN {X 0,Y 369.924,Z 426.353,A -85,B 0,C 180,E1 -16474.358,E2 -16474.358} C_VEL
LIN {X 0,Y 367.582,Z 425.054,A -85,B 0,C 180,E1 -16476.172,E2 -16476.172} C_VEL
LIN {X 0,Y 365.21,Z 423.141,A -85,B 0,C 180,E1 -16477.742,E2 -16477.742} C_VEL
LIN {X 0,Y 362.969,Z 420.853,A -85,B 0,C 180,E1 -16479.078,E2 -16479.078} C_VEL
LIN {X 0,Y 360.972,Z 418.907,A -85,B 0,C 180,E1 -16480.092,E2 -16480.092} C_VEL
LIN {X 0,Y 356.277,Z 415.48,A -85,B 0,C 180,E1 -16481.884,E2 -16481.884} C_VEL
LIN {X 0,Y 351.892,Z 411.284,A -85,B 0,C 180,E1 -16483.482,E2 -16483.482} C_VEL
LIN {X 0,Y 346.018,Z 406.017,A -85,B 0,C 180,E1 -16485.31,E2 -16485.31} C_VEL
LIN {X 0,Y 339.621,Z 399.777,A -85,B 0,C 180,E1 -16487.053,E2 -16487.053} C_VEL
LIN {X 0,Y 333.563,Z 393.566,A -85,B 0,C 180,E1 -16488.538,E2 -16488.538} C_VEL
LIN {X 0,Y 327.14,Z 386.614,A -85,B 0,C 180,E1 -16489.969,E2 -16489.969} C_VEL
LIN {X 0,Y 320.269,Z 378.649,A -85,B 0,C 180,E1 -16491.345,E2 -16491.345} C_VEL
LIN {X 0,Y 314.402,Z 371.306,A -85,B 0,C 180,E1 -16492.406,E2 -16492.406} C_VEL
LIN {X 0,Y 310.141,Z 365.745,A -85,B 0,C 180,E1 -16493.094,E2 -16493.094} C_VEL
LIN {X 0,Y 304.465,Z 357.333,A -85,B 0,C 180,E1 -16493.94,E2 -16493.94} C_VEL
LIN {X 0,Y 300.009,Z 348.759,A -85,B 0,C 180,E1 -16494.584,E2 -16494.584} C_VEL
LIN {X 0,Y 298.567,Z 345.358,A -85,B 0,C 180,E1 -16494.8,E2 -16494.8} C_VEL
LIN {X 0,Y 298.465,Z 344.808,A -85,B 0,C 180,E1 -16494.844,E2 -16494.844} C_VEL
LIN {X 0,Y 298.46,Z 344.809,A -85,B 0,C 180,E1 -16498.096,E2 -16498.096} C_VEL
LIN {X 0,Y 298.392,Z 344.818,A -85,B 0,C 180,E1 -16502.017,E2 -16502.017} C_VEL
LIN {X 0,Y 298.43,Z 344.813,A -85,B 0,C 180,E1 -16506.068,E2 -16506.068} C_VEL
LIN {X 0,Y 298.417,Z 344.812,A -85,B 0,C 180,E1 -16509.485,E2 -16509.485} C_VEL
LIN {X 0,Y 298.456,Z 344.805,A -85,B 0,C 180,E1 -16513.116,E2 -16513.116} C_VEL
LIN {X 0,Y 298.464,Z 344.805,A -85,B 0,C 180,E1 -16516.933,E2 -16516.933} C_VEL
LIN {X 0,Y 298.437,Z 344.809,A -85,B 0,C 180,E1 -16520.998,E2 -16520.998} C_VEL
LIN {X 0,Y 298.431,Z 344.812,A -85,B 0,C 180,E1 -16523.933,E2 -16523.933} C_VEL
LIN {X 0,Y 298.393,Z 344.815,A -85,B 0,C 180,E1 -16527.984,E2 -16527.984} C_VEL
LIN {X 0,Y 298.467,Z 344.806,A -85,B 0,C 180,E1 -16531.906,E2 -16531.906} C_VEL
LIN {X 0,Y 298.482,Z 344.802,A -85,B 0,C 180,E1 -16534.925,E2 -16534.925} C_VEL
LIN {X 0,Y 298.438,Z 344.81,A -85,B 0,C 180,E1 -16539.315,E2 -16539.315} C_VEL
LIN {X 0,Y 298.536,Z 344.796,A -85,B 0,C 180,E1 -16542.18,E2 -16542.18} C_VEL
LIN {X 0,Y 298.592,Z 344.791,A -85,B 0,C 180,E1 -16544.995,E2 -16544.995} C_VEL
LIN {X 0,Y 298.592,Z 344.791,A -85,B 0,C 180,E1 -16549.147,E2 -16549.147} C_VEL
LIN {X 0,Y 298.753,Z 344.768,A -85,B 0,C 180,E1 -16551.887,E2 -16551.887} C_VEL
LIN {X 0,Y 298.657,Z 344.783,A -85,B 0,C 180,E1 -16554.6,E2 -16554.6} C_VEL
LIN {X 0,Y 298.922,Z 344.739,A -85,B 0,C 180,E1 -16558.654,E2 -16558.654} C_VEL
LIN {X 0,Y 298.923,Z 344.747,A -85,B 0,C 180,E1 -16561.348,E2 -16561.348} C_VEL
LIN {X 0,Y 298.792,Z 344.768,A -85,B 0,C 180,E1 -16566.755,E2 -16566.755} C_VEL
LIN {X 0,Y 298.749,Z 344.77,A -85,B 0,C 180,E1 -16567.883,E2 -16567.883} C_VEL
LIN {X 0,Y 298.069,Z 344.858,A -85,B 0,C 180,E1 -16569.007,E2 -16569.007} C_VEL
LIN {X 0,Y 295.11,Z 345.226,A -85,B 0,C 180,E1 -16570.833,E2 -16570.833} C_VEL
LIN {X 0,Y 292.615,Z 345.537,A -85,B 0,C 180,E1 -16572.315,E2 -16572.315} C_VEL
LIN {X 0,Y 291.577,Z 345.664,A -85,B 0,C 180,E1 -16573.466,E2 -16573.466} C_VEL
LIN {X 0,Y 291.51,Z 345.673,A -85,B 0,C 180,E1 -16573.856,E2 -16573.856} C_VEL
LIN {X 0,Y 291.44,Z 345.682,A -85,B 0,C 180,E1 -16576.821,E2 -16576.821} C_VEL
LIN {X 0,Y 291.424,Z 345.683,A -85,B 0,C 180,E1 -16579.861,E2 -16579.861} C_VEL
LIN {X 0,Y 291.384,Z 345.692,A -85,B 0,C 180,E1 -16584.207,E2 -16584.207} C_VEL
LIN {X 0,Y 291.422,Z 345.684,A -85,B 0,C 180,E1 -16587.272,E2 -16587.272} C_VEL
LIN {X 0,Y 291.335,Z 345.697,A -85,B 0,C 180,E1 -16590.438,E2 -16590.438} C_VEL
LIN {X 0,Y 291.345,Z 345.699,A -85,B 0,C 180,E1 -16592.404,E2 -16592.404} C_VEL
LIN {X 0,Y 291.55,Z 347.108,A -85,B 0,C 180,E1 -16595.348,E2 -16595.348} C_VEL
LIN {X 0,Y 291.934,Z 349.784,A -85,B 0,C 180,E1 -16599.614,E2 -16599.614} C_VEL
LIN {X 0,Y 292.196,Z 351.638,A -85,B 0,C 180,E1 -16602.336,E2 -16602.336} C_VEL
LIN {X 0,Y 292.436,Z 354.475,A -85,B 0,C 180,E1 -16606.136,E2 -16606.136} C_VEL
LIN {X 0,Y 292.24,Z 357.233,A -85,B 0,C 180,E1 -16609.51,E2 -16609.51} C_VEL
LIN {X 0,Y 291.811,Z 360.253,A -85,B 0,C 180,E1 -16612.98,E2 -16612.98} C_VEL
LIN {X 0,Y 291.274,Z 363.315,A -85,B 0,C 180,E1 -16616.293,E2 -16616.293} C_VEL
LIN {X 0,Y 290.816,Z 366.35,A -85,B 0,C 180,E1 -16619.503,E2 -16619.503} C_VEL
LIN {X 0,Y 290.191,Z 370.969,A -85,B 0,C 180,E1 -16624.155,E2 -16624.155} C_VEL
LIN {X 0,Y 290.151,Z 371.645,A -85,B 0,C 180,E1 -16624.792,E2 -16624.792} C_VEL
LIN {X 0,Y 291.561,Z 377.077,A -85,B 0,C 180,E1 -16625.138,E2 -16625.138} C_VEL
LIN {X 0,Y 294.362,Z 388.619,A -85,B 0,C 180,E1 -16626.054,E2 -16626.054} C_VEL
LIN {X 0,Y 296.368,Z 399.412,A -85,B 0,C 180,E1 -16627.064,E2 -16627.064} C_VEL
LIN {X 0,Y 297.523,Z 408.857,A -85,B 0,C 180,E1 -16628.08,E2 -16628.08} C_VEL
LIN {X 0,Y 298.154,Z 417.308,A -85,B 0,C 180,E1 -16629.12,E2 -16629.12} C_VEL
LIN {X 0,Y 296.921,Z 426.209,A -85,B 0,C 180,E1 -16630.288,E2 -16630.288} C_VEL
LIN {X 0,Y 295.465,Z 434.737,A -85,B 0,C 180,E1 -16631.629,E2 -16631.629} C_VEL
LIN {X 0,Y 294.251,Z 442.567,A -85,B 0,C 180,E1 -16633.121,E2 -16633.121} C_VEL
LIN {X 0,Y 293.032,Z 449.539,A -85,B 0,C 180,E1 -16634.703,E2 -16634.703} C_VEL
LIN {X 0,Y 291.89,Z 455.855,A -85,B 0,C 180,E1 -16636.423,E2 -16636.423} C_VEL
LIN {X 0,Y 290.979,Z 461.117,A -85,B 0,C 180,E1 -16638.153,E2 -16638.153} C_VEL
LIN {X 0,Y 290.251,Z 466.25,A -85,B 0,C 180,E1 -16640.242,E2 -16640.242} C_VEL
LIN {X 0,Y 289.732,Z 470.24,A -85,B 0,C 180,E1 -16642.333,E2 -16642.333} C_VEL
LIN {X 0,Y 289.481,Z 473.293,A -85,B 0,C 180,E1 -16644.506,E2 -16644.506} C_VEL
LIN {X 0,Y 289.44,Z 475.644,A -85,B 0,C 180,E1 -16647.216,E2 -16647.216} C_VEL
LIN {X 0,Y 289.409,Z 476.233,A -85,B 0,C 180,E1 -16648.609,E2 -16648.609} C_VEL
LIN {X 0,Y 289.409,Z 476.233,A -85,B 0,C 180,E1 -16651.392,E2 -16651.392} C_VEL
LIN {X 0,Y 289.439,Z 475.644,A -85,B 0,C 180,E1 -16652.784,E2 -16652.784} C_VEL
LIN {X 0,Y 289.479,Z 473.192,A -85,B 0,C 180,E1 -16655.573,E2 -16655.573} C_VEL
LIN {X 0,Y 289.731,Z 470.24,A -85,B 0,C 180,E1 -16657.667,E2 -16657.667} C_VEL
LIN {X 0,Y 290.251,Z 466.25,A -85,B 0,C 180,E1 -16659.758,E2 -16659.758} C_VEL
LIN {X 0,Y 290.979,Z 461.117,A -85,B 0,C 180,E1 -16661.847,E2 -16661.847} C_VEL
LIN {X 0,Y 291.891,Z 455.855,A -85,B 0,C 180,E1 -16663.577,E2 -16663.577} C_VEL
LIN {X 0,Y 293.037,Z 449.539,A -85,B 0,C 180,E1 -16665.297,E2 -16665.297} C_VEL
LIN {X 0,Y 294.254,Z 442.573,A -85,B 0,C 180,E1 -16666.878,E2 -16666.878} C_VEL
LIN {X 0,Y 295.45,Z 434.737,A -85,B 0,C 180,E1 -16668.372,E2 -16668.372} C_VEL
LIN {X 0,Y 296.902,Z 426.209,A -85,B 0,C 180,E1 -16669.713,E2 -16669.713} C_VEL
LIN {X 0,Y 298.141,Z 417.304,A -85,B 0,C 180,E1 -16670.882,E2 -16670.882} C_VEL
LIN {X 0,Y 297.239,Z 406.28,A -85,B 0,C 180,E1 -16672.229,E2 -16672.229} C_VEL
LIN {X 0,Y 295.481,Z 393.823,A -85,B 0,C 180,E1 -16673.478,E2 -16673.478} C_VEL
LIN {X 0,Y 292.972,Z 382.43,A -85,B 0,C 180,E1 -16674.447,E2 -16674.447} C_VEL
LIN {X 0,Y 290.239,Z 372.552,A -85,B 0,C 180,E1 -16675.167,E2 -16675.167} C_VEL
LIN {X 0,Y 290.146,Z 371.584,A -85,B 0,C 180,E1 -16675.24,E2 -16675.24} C_VEL
LIN {X 0,Y 290.69,Z 367.298,A -85,B 0,C 180,E1 -16679.497,E2 -16679.497} C_VEL
LIN {X 0,Y 291.106,Z 364.566,A -85,B 0,C 180,E1 -16682.328,E2 -16682.328} C_VEL
LIN {X 0,Y 291.52,Z 361.733,A -85,B 0,C 180,E1 -16685.352,E2 -16685.352} C_VEL
LIN {X 0,Y 292.03,Z 358.716,A -85,B 0,C 180,E1 -16688.735,E2 -16688.735} C_VEL
LIN {X 0,Y 292.378,Z 355.699,A -85,B 0,C 180,E1 -16692.302,E2 -16692.302} C_VEL
LIN {X 0,Y 292.427,Z 354.209,A -85,B 0,C 180,E1 -16694.184,E2 -16694.184} C_VEL
LIN {X 0,Y 292.188,Z 351.637,A -85,B 0,C 180,E1 -16697.662,E2 -16697.662} C_VEL
LIN {X 0,Y 291.844,Z 349.214,A -85,B 0,C 180,E1 -16701.235,E2 -16701.235} C_VEL
LIN {X 0,Y 291.528,Z 346.871,A -85,B 0,C 180,E1 -16705.05,E2 -16705.05} C_VEL
LIN {X 0,Y 291.345,Z 345.7,A -85,B 0,C 180,E1 -16707.596,E2 -16707.596} C_VEL
LIN {X 0,Y 291.379,Z 345.69,A -85,B 0,C 180,E1 -16711.157,E2 -16711.157} C_VEL
LIN {X 0,Y 291.416,Z 345.685,A -85,B 0,C 180,E1 -16714.271,E2 -16714.271} C_VEL
LIN {X 0,Y 291.373,Z 345.691,A -85,B 0,C 180,E1 -16717.298,E2 -16717.298} C_VEL
LIN {X 0,Y 291.44,Z 345.681,A -85,B 0,C 180,E1 -16720.268,E2 -16720.268} C_VEL
LIN {X 0,Y 291.498,Z 345.673,A -85,B 0,C 180,E1 -16724.665,E2 -16724.665} C_VEL
LIN {X 0,Y 291.537,Z 345.669,A -85,B 0,C 180,E1 -16728.88,E2 -16728.88} C_VEL
LIN {X 0,Y 291.706,Z 345.649,A -85,B 0,C 180,E1 -16731.688,E2 -16731.688} C_VEL
LIN {X 0,Y 291.628,Z 345.656,A -85,B 0,C 180,E1 -16734.468,E2 -16734.468} C_VEL
LIN {X 0,Y 291.889,Z 345.623,A -85,B 0,C 180,E1 -16738.62,E2 -16738.62} C_VEL
LIN {X 0,Y 291.888,Z 345.614,A -85,B 0,C 180,E1 -16741.379,E2 -16741.379} C_VEL
LIN {X 0,Y 291.74,Z 345.646,A -85,B 0,C 180,E1 -16746.917,E2 -16746.917} C_VEL
LIN {X 0,Y 291.628,Z 345.654,A -85,B 0,C 180,E1 -16749.711,E2 -16749.711} C_VEL
LIN {X 0,Y 291.521,Z 345.668,A -85,B 0,C 180,E1 -16753.95,E2 -16753.95} C_VEL
LIN {X 0,Y 291.485,Z 345.679,A -85,B 0,C 180,E1 -16756.817,E2 -16756.817} C_VEL
LIN {X 0,Y 291.449,Z 345.676,A -85,B 0,C 180,E1 -16759.874,E2 -16759.874} C_VEL
LIN {X 0,Y 291.381,Z 345.688,A -85,B 0,C 180,E1 -16764.206,E2 -16764.206} C_VEL
LIN {X 0,Y 291.423,Z 345.682,A -85,B 0,C 180,E1 -16767.27,E2 -16767.27} C_VEL
LIN {X 0,Y 291.335,Z 345.697,A -85,B 0,C 180,E1 -16770.436,E2 -16770.436} C_VEL
LIN {X 0,Y 291.342,Z 345.692,A -85,B 0,C 180,E1 -16773.698,E2 -16773.698} C_VEL
LIN {X 0,Y 291.402,Z 345.685,A -85,B 0,C 180,E1 -16777.261,E2 -16777.261} C_VEL
LIN {X 0,Y 291.402,Z 345.686,A -85,B 0,C 180,E1 -16780.63,E2 -16780.63} C_VEL
LIN {X 0,Y 291.351,Z 345.693,A -85,B 0,C 180,E1 -16784.389,E2 -16784.389} C_VEL
LIN {X 0,Y 291.354,Z 345.692,A -85,B 0,C 180,E1 -16788.397,E2 -16788.397} C_VEL
LIN {X 0,Y 291.377,Z 345.688,A -85,B 0,C 180,E1 -16791.162,E2 -16791.162} C_VEL
LIN {X 0,Y 291.382,Z 345.688,A -85,B 0,C 180,E1 -16794.629,E2 -16794.629} C_VEL
LIN {X 0,Y 291.369,Z 345.693,A -85,B 0,C 180,E1 -16797.951,E2 -16797.951} C_VEL
LIN {X 0,Y 291.379,Z 345.69,A -85,B 0,C 180,E1 -16801.158,E2 -16801.158} C_VEL
LIN {X 0,Y 291.44,Z 345.682,A -85,B 0,C 180,E1 -16804.533,E2 -16804.533} C_VEL
LIN {X 0,Y 292.474,Z 348.559,A -85,B 0,C 180,E1 -16804.728,E2 -16804.728} C_VEL
LIN {X 0,Y 297.364,Z 358.645,A -85,B 0,C 180,E1 -16805.497,E2 -16805.497} C_VEL
LIN {X 0,Y 302.567,Z 367.229,A -85,B 0,C 180,E1 -16806.353,E2 -16806.353} C_VEL
LIN {X 0,Y 308.188,Z 374.907,A -85,B 0,C 180,E1 -16807.282,E2 -16807.282} C_VEL
LIN {X 0,Y 315.247,Z 383.635,A -85,B 0,C 180,E1 -16808.54,E2 -16808.54} C_VEL
LIN {X 0,Y 321.848,Z 391.304,A -85,B 0,C 180,E1 -16809.876,E2 -16809.876} C_VEL
LIN {X 0,Y 328.112,Z 398.107,A -85,B 0,C 180,E1 -16811.259,E2 -16811.259} C_VEL
LIN {X 0,Y 333.486,Z 403.645,A -85,B 0,C 180,E1 -16812.552,E2 -16812.552} C_VEL
LIN {X 0,Y 338.947,Z 408.778,A -85,B 0,C 180,E1 -16813.973,E2 -16813.973} C_VEL
LIN {X 0,Y 343.403,Z 413.393,A -85,B 0,C 180,E1 -16815.336,E2 -16815.336} C_VEL
LIN {X 0,Y 348.13,Z 417.516,A -85,B 0,C 180,E1 -16816.845,E2 -16816.845} C_VEL
LIN {X 0,Y 352.634,Z 421.654,A -85,B 0,C 180,E1 -16818.504,E2 -16818.504} C_VEL
LIN {X 0,Y 356.695,Z 424.615,A -85,B 0,C 180,E1 -16820.111,E2 -16820.111} C_VEL
LIN {X 0,Y 360.304,Z 428.245,A -85,B 0,C 180,E1 -16822.152,E2 -16822.152} C_VEL
LIN {X 0,Y 362.101,Z 429.782,A -85,B 0,C 180,E1 -16823.313,E2 -16823.313} C_VEL
LIN {X 0,Y 363.709,Z 430.884,A -85,B 0,C 180,E1 -16824.456,E2 -16824.456} C_VEL
LIN {X 0,Y 366.147,Z 432.002,A -85,B 0,C 180,E1 -16826.467,E2 -16826.467} C_VEL
LIN {X 0,Y 367.351,Z 432.318,A -85,B 0,C 180,E1 -16827.807,E2 -16827.807} C_VEL
LIN {X 0,Y 367.939,Z 432.452,A -85,B 0,C 180,E1 -16828.906,E2 -16828.906} C_VEL
LIN {X 0,Y 368.147,Z 432.485,A -85,B 0,C 180,E1 -16830,E2 -16830} C_VEL
LIN {X 0,Y 367.939,Z 432.451,A -85,B 0,C 180,E1 -16831.094,E2 -16831.094} C_VEL
LIN {X 0,Y 367.335,Z 432.328,A -85,B 0,C 180,E1 -16832.193,E2 -16832.193} C_VEL
LIN {X 0,Y 366.147,Z 431.997,A -85,B 0,C 180,E1 -16833.533,E2 -16833.533} C_VEL
LIN {X 0,Y 363.724,Z 430.894,A -85,B 0,C 180,E1 -16835.544,E2 -16835.544} C_VEL
LIN {X 0,Y 361.291,Z 429.123,A -85,B 0,C 180,E1 -16837.223,E2 -16837.223} C_VEL
LIN {X 0,Y 358.352,Z 426.248,A -85,B 0,C 180,E1 -16839.027,E2 -16839.027} C_VEL
LIN {X 0,Y 355.922,Z 423.998,A -85,B 0,C 180,E1 -16840.237,E2 -16840.237} C_VEL
LIN {X 0,Y 351.811,Z 420.999,A -85,B 0,C 180,E1 -16841.807,E2 -16841.807} C_VEL
LIN {X 0,Y 347.003,Z 416.433,A -85,B 0,C 180,E1 -16843.554,E2 -16843.554} C_VEL
LIN {X 0,Y 342.092,Z 412.085,A -85,B 0,C 180,E1 -16845.08,E2 -16845.08} C_VEL
LIN {X 0,Y 337.161,Z 407.242,A -85,B 0,C 180,E1 -16846.496,E2 -16846.496} C_VEL
LIN {X 0,Y 330.797,Z 400.797,A -85,B 0,C 180,E1 -16848.121,E2 -16848.121} C_VEL
LIN {X 0,Y 324.805,Z 394.397,A -85,B 0,C 180,E1 -16849.509,E2 -16849.509} C_VEL
LIN {X 0,Y 318.133,Z 386.96,A -85,B 0,C 180,E1 -16850.904,E2 -16850.904} C_VEL
LIN {X 0,Y 311.187,Z 378.791,A -85,B 0,C 180,E1 -16852.188,E2 -16852.188} C_VEL
LIN {X 0,Y 304.662,Z 370.092,A -85,B 0,C 180,E1 -16853.309,E2 -16853.309} C_VEL
LIN {X 0,Y 298.655,Z 361.017,A -85,B 0,C 180,E1 -16854.289,E2 -16854.289} C_VEL
LIN {X 0,Y 294.314,Z 352.515,A -85,B 0,C 180,E1 -16854.99,E2 -16854.99} C_VEL
LIN {X 0,Y 291.617,Z 346.664,A -85,B 0,C 180,E1 -16855.403,E2 -16855.403} C_VEL
LIN {X 0,Y 291.43,Z 345.683,A -85,B 0,C 180,E1 -16855.497,E2 -16855.497} C_VEL
LIN {X 0,Y 291.379,Z 345.69,A -85,B 0,C 180,E1 -16858.842,E2 -16858.842} C_VEL
LIN {X 0,Y 291.341,Z 345.696,A -85,B 0,C 180,E1 -16862.404,E2 -16862.404} C_VEL
LIN {X 0,Y 291.382,Z 345.688,A -85,B 0,C 180,E1 -16865.371,E2 -16865.371} C_VEL
LIN {X 0,Y 291.377,Z 345.688,A -85,B 0,C 180,E1 -16868.838,E2 -16868.838} C_VEL
LIN {X 0,Y 291.351,Z 345.692,A -85,B 0,C 180,E1 -16872.487,E2 -16872.487} C_VEL
LIN {X 0,Y 291.368,Z 345.69,A -85,B 0,C 180,E1 -16876.354,E2 -16876.354} C_VEL
LIN {X 0,Y 291.41,Z 345.684,A -85,B 0,C 180,E1 -16880.511,E2 -16880.511} C_VEL
LIN {X 0,Y 291.431,Z 345.681,A -85,B 0,C 180,E1 -16882.924,E2 -16882.924} C_VEL
LIN {X 0,Y 291.342,Z 345.692,A -85,B 0,C 180,E1 -16886.302,E2 -16886.302} C_VEL
LIN {X 0,Y 291.385,Z 345.687,A -85,B 0,C 180,E1 -16890.261,E2 -16890.261} C_VEL
LIN {X 0,Y 291.417,Z 345.681,A -85,B 0,C 180,E1 -16894.273,E2 -16894.273} C_VEL
LIN {X 0,Y 291.372,Z 345.692,A -85,B 0,C 180,E1 -16897.3,E2 -16897.3} C_VEL
LIN {X 0,Y 291.456,Z 345.675,A -85,B 0,C 180,E1 -16900.271,E2 -16900.271} C_VEL
LIN {X 0,Y 291.554,Z 345.665,A -85,B 0,C 180,E1 -16904.624,E2 -16904.624} C_VEL
LIN {X 0,Y 291.536,Z 345.671,A -85,B 0,C 180,E1 -16908.881,E2 -16908.881} C_VEL
LIN {X 0,Y 291.705,Z 345.647,A -85,B 0,C 180,E1 -16911.689,E2 -16911.689} C_VEL
LIN {X 0,Y 291.627,Z 345.657,A -85,B 0,C 180,E1 -16914.469,E2 -16914.469} C_VEL
LIN {X 0,Y 291.888,Z 345.614,A -85,B 0,C 180,E1 -16918.621,E2 -16918.621} C_VEL
LIN {X 0,Y 291.889,Z 345.623,A -85,B 0,C 180,E1 -16921.38,E2 -16921.38} C_VEL
LIN {X 0,Y 291.741,Z 345.645,A -85,B 0,C 180,E1 -16926.919,E2 -16926.919} C_VEL
LIN {X 0,Y 291.629,Z 345.657,A -85,B 0,C 180,E1 -16929.713,E2 -16929.713} C_VEL
LIN {X 0,Y 291.51,Z 345.673,A -85,B 0,C 180,E1 -16933.856,E2 -16933.856} C_VEL
LIN {X 0,Y 290.869,Z 345.756,A -85,B 0,C 180,E1 -16935.009,E2 -16935.009} C_VEL
LIN {X 0,Y 287.951,Z 346.117,A -85,B 0,C 180,E1 -16936.882,E2 -16936.882} C_VEL
LIN {X 0,Y 285.471,Z 346.428,A -85,B 0,C 180,E1 -16938.405,E2 -16938.405} C_VEL
LIN {X 0,Y 284.437,Z 346.553,A -85,B 0,C 180,E1 -16939.586,E2 -16939.586} C_VEL
LIN {X 0,Y 284.371,Z 346.563,A -85,B 0,C 180,E1 -16939.986,E2 -16939.986} C_VEL
LIN {X 0,Y 284.335,Z 346.568,A -85,B 0,C 180,E1 -16943.86,E2 -16943.86} C_VEL
LIN {X 0,Y 284.397,Z 346.559,A -85,B 0,C 180,E1 -16947.174,E2 -16947.174} C_VEL
LIN {X 0,Y 284.295,Z 346.575,A -85,B 0,C 180,E1 -16951.275,E2 -16951.275} C_VEL
LIN {X 0,Y 284.339,Z 346.859,A -85,B 0,C 180,E1 -16952.942,E2 -16952.942} C_VEL
LIN {X 0,Y 284.588,Z 348.789,A -85,B 0,C 180,E1 -16956.349,E2 -16956.349} C_VEL
LIN {X 0,Y 284.962,Z 351.147,A -85,B 0,C 180,E1 -16960.133,E2 -16960.133} C_VEL
LIN {X 0,Y 285.255,Z 353.533,A -85,B 0,C 180,E1 -16963.619,E2 -16963.619} C_VEL
LIN {X 0,Y 285.363,Z 355.596,A -85,B 0,C 180,E1 -16966.402,E2 -16966.402} C_VEL
LIN {X 0,Y 285.159,Z 358.329,A -85,B 0,C 180,E1 -16969.821,E2 -16969.821} C_VEL
LIN {X 0,Y 284.606,Z 361.639,A -85,B 0,C 180,E1 -16973.655,E2 -16973.655} C_VEL
LIN {X 0,Y 284.07,Z 364.901,A -85,B 0,C 180,E1 -16977.265,E2 -16977.265} C_VEL
LIN {X 0,Y 283.616,Z 367.745,A -85,B 0,C 180,E1 -16980.291,E2 -16980.291} C_VEL
LIN {X 0,Y 283.126,Z 371.417,A -85,B 0,C 180,E1 -16984.1,E2 -16984.1} C_VEL
LIN {X 0,Y 286.932,Z 386.106,A -85,B 0,C 180,E1 -16985.224,E2 -16985.224} C_VEL
LIN {X 0,Y 289.347,Z 398.498,A -85,B 0,C 180,E1 -16986.408,E2 -16986.408} C_VEL
LIN {X 0,Y 290.609,Z 408.596,A -85,B 0,C 180,E1 -16987.524,E2 -16987.524} C_VEL
LIN {X 0,Y 291.281,Z 417.215,A -85,B 0,C 180,E1 -16988.618,E2 -16988.618} C_VEL
LIN {X 0,Y 290.852,Z 422.476,A -85,B 0,C 180,E1 -16989.305,E2 -16989.305} C_VEL
LIN {X 0,Y 289.077,Z 432.622,A -85,B 0,C 180,E1 -16990.84,E2 -16990.84} C_VEL
LIN {X 0,Y 287.657,Z 440.657,A -85,B 0,C 180,E1 -16992.336,E2 -16992.336} C_VEL
LIN {X 0,Y 286.397,Z 447.965,A -85,B 0,C 180,E1 -16993.974,E2 -16993.974} C_VEL
LIN {X 0,Y 285.182,Z 454.503,A -85,B 0,C 180,E1 -16995.733,E2 -16995.733} C_VEL
LIN {X 0,Y 284.324,Z 459.004,A -85,B 0,C 180,E1 -16997.146,E2 -16997.146} C_VEL
LIN {X 0,Y 283.441,Z 464.498,A -85,B 0,C 180,E1 -16999.283,E2 -16999.283} C_VEL
LIN {X 0,Y 282.828,Z 468.826,A -85,B 0,C 180,E1 -17001.426,E2 -17001.426} C_VEL
LIN {X 0,Y 282.576,Z 471.195,A -85,B 0,C 180,E1 -17002.856,E2 -17002.856} C_VEL
LIN {X 0,Y 282.373,Z 473.398,A -85,B 0,C 180,E1 -17004.608,E2 -17004.608} C_VEL
LIN {X 0,Y 282.347,Z 475.448,A -85,B 0,C 180,E1 -17007.146,E2 -17007.146} C_VEL
LIN {X 0,Y 282.332,Z 476.038,A -85,B 0,C 180,E1 -17008.574,E2 -17008.574} C_VEL
LIN {X 0,Y 282.332,Z 476.038,A -85,B 0,C 180,E1 -17011.426,E2 -17011.426} C_VEL
LIN {X 0,Y 282.346,Z 475.448,A -85,B 0,C 180,E1 -17012.854,E2 -17012.854} C_VEL
LIN {X 0,Y 282.388,Z 472.996,A -85,B 0,C 180,E1 -17015.713,E2 -17015.713} C_VEL
LIN {X 0,Y 282.687,Z 470.044,A -85,B 0,C 180,E1 -17017.859,E2 -17017.859} C_VEL
LIN {X 0,Y 283.216,Z 466.053,A -85,B 0,C 180,E1 -17020.003,E2 -17020.003} C_VEL
LIN {X 0,Y 283.982,Z 460.92,A -85,B 0,C 180,E1 -17022.143,E2 -17022.143} C_VEL
LIN {X 0,Y 284.974,Z 455.659,A -85,B 0,C 180,E1 -17023.913,E2 -17023.913} C_VEL
LIN {X 0,Y 286.142,Z 449.341,A -85,B 0,C 180,E1 -17025.674,E2 -17025.674} C_VEL
LIN {X 0,Y 287.271,Z 443.391,A -85,B 0,C 180,E1 -17027.072,E2 -17027.072} C_VEL
LIN {X 0,Y 288.367,Z 436.46,A -85,B 0,C 180,E1 -17028.471,E2 -17028.471} C_VEL
LIN {X 0,Y 289.803,Z 428.281,A -85,B 0,C 180,E1 -17029.847,E2 -17029.847} C_VEL
LIN {X 0,Y 291.243,Z 419.772,A -85,B 0,C 180,E1 -17031.036,E2 -17031.036} C_VEL
LIN {X 0,Y 290.92,Z 411.935,A -85,B 0,C 180,E1 -17032.071,E2 -17032.071} C_VEL
LIN {X 0,Y 289.971,Z 402.584,A -85,B 0,C 180,E1 -17033.158,E2 -17033.158} C_VEL
LIN {X 0,Y 288.321,Z 392.467,A -85,B 0,C 180,E1 -17034.181,E2 -17034.181} C_VEL
LIN {X 0,Y 285.948,Z 382.079,A -85,B 0,C 180,E1 -17035.097,E2 -17035.097} C_VEL
LIN {X 0,Y 283.127,Z 371.423,A -85,B 0,C 180,E1 -17035.898,E2 -17035.898} C_VEL
LIN {X 0,Y 283.669,Z 367.529,A -85,B 0,C 180,E1 -17039.871,E2 -17039.871} C_VEL
LIN {X 0,Y 284.097,Z 364.645,A -85,B 0,C 180,E1 -17042.972,E2 -17042.972} C_VEL
LIN {X 0,Y 284.603,Z 361.6,A -85,B 0,C 180,E1 -17046.346,E2 -17046.346} C_VEL
LIN {X 0,Y 285.159,Z 358.328,A -85,B 0,C 180,E1 -17050.179,E2 -17050.179} C_VEL
LIN {X 0,Y 285.361,Z 355.585,A -85,B 0,C 180,E1 -17053.598,E2 -17053.598} C_VEL
LIN {X 0,Y 285.252,Z 353.531,A -85,B 0,C 180,E1 -17056.38,E2 -17056.38} C_VEL
LIN {X 0,Y 284.931,Z 350.986,A -85,B 0,C 180,E1 -17060.11,E2 -17060.11} C_VEL
LIN {X 0,Y 284.587,Z 348.786,A -85,B 0,C 180,E1 -17063.651,E2 -17063.651} C_VEL
LIN {X 0,Y 284.318,Z 346.792,A -85,B 0,C 180,E1 -17067.186,E2 -17067.186} C_VEL
LIN {X 0,Y 284.357,Z 346.566,A -85,B 0,C 180,E1 -17070.375,E2 -17070.375} C_VEL
LIN {X 0,Y 284.378,Z 346.564,A -85,B 0,C 180,E1 -17073.586,E2 -17073.586} C_VEL
LIN {X 0,Y 284.334,Z 346.567,A -85,B 0,C 180,E1 -17076.703,E2 -17076.703} C_VEL
LIN {X 0,Y 284.377,Z 346.564,A -85,B 0,C 180,E1 -17079.904,E2 -17079.904} C_VEL
LIN {X 0,Y 284.448,Z 346.551,A -85,B 0,C 180,E1 -17084.491,E2 -17084.491} C_VEL
LIN {X 0,Y 284.488,Z 346.546,A -85,B 0,C 180,E1 -17088.601,E2 -17088.601} C_VEL
LIN {X 0,Y 284.657,Z 346.529,A -85,B 0,C 180,E1 -17091.48,E2 -17091.48} C_VEL
LIN {X 0,Y 284.598,Z 346.532,A -85,B 0,C 180,E1 -17094.33,E2 -17094.33} C_VEL
LIN {X 0,Y 284.855,Z 346.499,A -85,B 0,C 180,E1 -17098.585,E2 -17098.585} C_VEL
LIN {X 0,Y 284.854,Z 346.488,A -85,B 0,C 180,E1 -17101.413,E2 -17101.413} C_VEL
LIN {X 0,Y 284.693,Z 346.524,A -85,B 0,C 180,E1 -17107.089,E2 -17107.089} C_VEL
LIN {X 0,Y 284.565,Z 346.533,A -85,B 0,C 180,E1 -17109.955,E2 -17109.955} C_VEL
LIN {X 0,Y 284.48,Z 346.546,A -85,B 0,C 180,E1 -17114.302,E2 -17114.302} C_VEL
LIN {X 0,Y 284.424,Z 346.555,A -85,B 0,C 180,E1 -17117.248,E2 -17117.248} C_VEL
LIN {X 0,Y 284.375,Z 346.558,A -85,B 0,C 180,E1 -17120.242,E2 -17120.242} C_VEL
LIN {X 0,Y 284.338,Z 346.565,A -85,B 0,C 180,E1 -17124.846,E2 -17124.846} C_VEL
LIN {X 0,Y 284.332,Z 346.567,A -85,B 0,C 180,E1 -17128.01,E2 -17128.01} C_VEL
LIN {X 0,Y 284.294,Z 346.57,A -85,B 0,C 180,E1 -17131.274,E2 -17131.274} C_VEL
LIN {X 0,Y 284.359,Z 346.562,A -85,B 0,C 180,E1 -17135.353,E2 -17135.353} C_VEL
LIN {X 0,Y 284.335,Z 346.568,A -85,B 0,C 180,E1 -17138.164,E2 -17138.164} C_VEL
LIN {X 0,Y 284.34,Z 346.568,A -85,B 0,C 180,E1 -17142.14,E2 -17142.14} C_VEL
LIN {X 0,Y 284.316,Z 346.571,A -85,B 0,C 180,E1 -17146.201,E2 -17146.201} C_VEL
LIN {X 0,Y 284.348,Z 346.567,A -85,B 0,C 180,E1 -17150.013,E2 -17150.013} C_VEL
LIN {X 0,Y 284.351,Z 346.566,A -85,B 0,C 180,E1 -17153.617,E2 -17153.617} C_VEL
LIN {X 0,Y 284.304,Z 346.57,A -85,B 0,C 180,E1 -17157.189,E2 -17157.189} C_VEL
LIN {X 0,Y 284.355,Z 346.564,A -85,B 0,C 180,E1 -17160.376,E2 -17160.376} C_VEL
LIN {X 0,Y 284.377,Z 346.563,A -85,B 0,C 180,E1 -17163.891,E2 -17163.891} C_VEL
LIN {X 0,Y 285.391,Z 349.447,A -85,B 0,C 180,E1 -17164.073,E2 -17164.073} C_VEL
LIN {X 0,Y 291.671,Z 362.455,A -85,B 0,C 180,E1 -17165.143,E2 -17165.143} C_VEL
LIN {X 0,Y 296.948,Z 371.39,A -85,B 0,C 180,E1 -17166.116,E2 -17166.116} C_VEL
LIN {X 0,Y 304.365,Z 381.407,A -85,B 0,C 180,E1 -17167.46,E2 -17167.46} C_VEL
LIN {X 0,Y 311.88,Z 390.553,A -85,B 0,C 180,E1 -17168.866,E2 -17168.866} C_VEL
LIN {X 0,Y 319.229,Z 398.824,A -85,B 0,C 180,E1 -17170.394,E2 -17170.394} C_VEL
LIN {X 0,Y 325.44,Z 405.431,A -85,B 0,C 180,E1 -17171.839,E2 -17171.839} C_VEL
LIN {X 0,Y 330.473,Z 410.713,A -85,B 0,C 180,E1 -17173.132,E2 -17173.132} C_VEL
LIN {X 0,Y 335.511,Z 415.461,A -85,B 0,C 180,E1 -17174.484,E2 -17174.484} C_VEL
LIN {X 0,Y 341.271,Z 420.877,A -85,B 0,C 180,E1 -17176.276,E2 -17176.276} C_VEL
LIN {X 0,Y 346.96,Z 426.097,A -85,B 0,C 180,E1 -17178.313,E2 -17178.313} C_VEL
LIN {X 0,Y 350.314,Z 428.637,A -85,B 0,C 180,E1 -17179.598,E2 -17179.598} C_VEL
LIN {X 0,Y 352.932,Z 430.83,A -85,B 0,C 180,E1 -17180.833,E2 -17180.833} C_VEL
LIN {X 0,Y 354.931,Z 432.912,A -85,B 0,C 180,E1 -17182.033,E2 -17182.033} C_VEL
LIN {X 0,Y 356.797,Z 434.514,A -85,B 0,C 180,E1 -17183.213,E2 -17183.213} C_VEL
LIN {X 0,Y 359.644,Z 436.383,A -85,B 0,C 180,E1 -17185.277,E2 -17185.277} C_VEL
LIN {X 0,Y 361.26,Z 437.029,A -85,B 0,C 180,E1 -17186.654,E2 -17186.654} C_VEL
LIN {X 0,Y 362.273,Z 437.317,A -85,B 0,C 180,E1 -17187.776,E2 -17187.776} C_VEL
LIN {X 0,Y 362.907,Z 437.453,A -85,B 0,C 180,E1 -17188.89,E2 -17188.89} C_VEL
LIN {X 0,Y 363.131,Z 437.486,A -85,B 0,C 180,E1 -17190,E2 -17190} C_VEL
LIN {X 0,Y 362.906,Z 437.455,A -85,B 0,C 180,E1 -17191.11,E2 -17191.11} C_VEL
LIN {X 0,Y 362.254,Z 437.328,A -85,B 0,C 180,E1 -17192.224,E2 -17192.224} C_VEL
LIN {X 0,Y 361.259,Z 437.025,A -85,B 0,C 180,E1 -17193.346,E2 -17193.346} C_VEL
LIN {X 0,Y 359.644,Z 436.399,A -85,B 0,C 180,E1 -17194.723,E2 -17194.723} C_VEL
LIN {X 0,Y 356.752,Z 434.538,A -85,B 0,C 180,E1 -17196.788,E2 -17196.788} C_VEL
LIN {X 0,Y 354.862,Z 432.827,A -85,B 0,C 180,E1 -17198.016,E2 -17198.016} C_VEL
LIN {X 0,Y 352.087,Z 430.029,A -85,B 0,C 180,E1 -17199.611,E2 -17199.611} C_VEL
LIN {X 0,Y 348.654,Z 427.477,A -85,B 0,C 180,E1 -17201.02,E2 -17201.02} C_VEL
LIN {X 0,Y 343.398,Z 422.794,A -85,B 0,C 180,E1 -17203.01,E2 -17203.01} C_VEL
LIN {X 0,Y 337.575,Z 417.564,A -85,B 0,C 180,E1 -17204.879,E2 -17204.879} C_VEL
LIN {X 0,Y 331.866,Z 411.981,A -85,B 0,C 180,E1 -17206.52,E2 -17206.52} C_VEL
LIN {X 0,Y 325.442,Z 405.467,A -85,B 0,C 180,E1 -17208.162,E2 -17208.162} C_VEL
LIN {X 0,Y 318.092,Z 397.652,A -85,B 0,C 180,E1 -17209.839,E2 -17209.839} C_VEL
LIN {X 0,Y 311.232,Z 389.914,A -85,B 0,C 180,E1 -17211.248,E2 -17211.248} C_VEL
LIN {X 0,Y 303.013,Z 379.713,A -85,B 0,C 180,E1 -17212.789,E2 -17212.789} C_VEL
LIN {X 0,Y 295.759,Z 369.493,A -85,B 0,C 180,E1 -17214.11,E2 -17214.11} C_VEL
LIN {X 0,Y 290.674,Z 360.583,A -85,B 0,C 180,E1 -17215.031,E2 -17215.031} C_VEL
LIN {X 0,Y 284.531,Z 347.442,A -85,B 0,C 180,E1 -17216.067,E2 -17216.067} C_VEL
LIN {X 0,Y 284.382,Z 346.563,A -85,B 0,C 180,E1 -17216.135,E2 -17216.135} C_VEL
LIN {X 0,Y 284.311,Z 346.572,A -85,B 0,C 180,E1 -17220.099,E2 -17220.099} C_VEL
LIN {X 0,Y 284.302,Z 346.57,A -85,B 0,C 180,E1 -17222.945,E2 -17222.945} C_VEL
LIN {X 0,Y 284.351,Z 346.566,A -85,B 0,C 180,E1 -17226.383,E2 -17226.383} C_VEL
LIN {X 0,Y 284.348,Z 346.567,A -85,B 0,C 180,E1 -17229.987,E2 -17229.987} C_VEL
LIN {X 0,Y 284.306,Z 346.571,A -85,B 0,C 180,E1 -17234.204,E2 -17234.204} C_VEL
LIN {X 0,Y 284.337,Z 346.567,A -85,B 0,C 180,E1 -17238.137,E2 -17238.137} C_VEL
LIN {X 0,Y 284.343,Z 346.565,A -85,B 0,C 180,E1 -17242.272,E2 -17242.272} C_VEL
LIN {X 0,Y 284.321,Z 346.569,A -85,B 0,C 180,E1 -17245.354,E2 -17245.354} C_VEL
LIN {X 0,Y 284.294,Z 346.57,A -85,B 0,C 180,E1 -17248.726,E2 -17248.726} C_VEL
LIN {X 0,Y 284.397,Z 346.558,A -85,B 0,C 180,E1 -17252.826,E2 -17252.826} C_VEL
LIN {X 0,Y 284.331,Z 346.565,A -85,B 0,C 180,E1 -17256.705,E2 -17256.705} C_VEL
LIN {X 0,Y 284.402,Z 346.558,A -85,B 0,C 180,E1 -17261.262,E2 -17261.262} C_VEL
LIN {X 0,Y 284.491,Z 346.545,A -85,B 0,C 180,E1 -17264.46,E2 -17264.46} C_VEL
LIN {X 0,Y 284.487,Z 346.547,A -85,B 0,C 180,E1 -17268.602,E2 -17268.602} C_VEL
LIN {X 0,Y 284.656,Z 346.526,A -85,B 0,C 180,E1 -17271.482,E2 -17271.482} C_VEL
LIN {X 0,Y 284.598,Z 346.532,A -85,B 0,C 180,E1 -17274.332,E2 -17274.332} C_VEL
LIN {X 0,Y 284.854,Z 346.488,A -85,B 0,C 180,E1 -17278.587,E2 -17278.587} C_VEL
LIN {X 0,Y 284.855,Z 346.499,A -85,B 0,C 180,E1 -17281.415,E2 -17281.415} C_VEL
LIN {X 0,Y 284.694,Z 346.522,A -85,B 0,C 180,E1 -17287.091,E2 -17287.091} C_VEL
LIN {X 0,Y 284.567,Z 346.537,A -85,B 0,C 180,E1 -17289.956,E2 -17289.956} C_VEL
LIN {X 0,Y 284.464,Z 346.553,A -85,B 0,C 180,E1 -17294.304,E2 -17294.304} C_VEL
LIN {X 0,Y 284.374,Z 346.562,A -85,B 0,C 180,E1 -17298.741,E2 -17298.741} C_VEL
LIN {X 0,Y 284.371,Z 346.563,A -85,B 0,C 180,E1 -17299.986,E2 -17299.986} C_VEL
LIN {X 0,Y 283.741,Z 346.647,A -85,B 0,C 180,E1 -17301.169,E2 -17301.169} C_VEL
LIN {X 0,Y 280.868,Z 347.005,A -85,B 0,C 180,E1 -17303.094,E2 -17303.094} C_VEL
LIN {X 0,Y 278.415,Z 347.306,A -85,B 0,C 180,E1 -17304.658,E2 -17304.658} C_VEL
LIN {X 0,Y 277.379,Z 347.436,A -85,B 0,C 180,E1 -17305.872,E2 -17305.872} C_VEL
LIN {X 0,Y 277.306,Z 347.44,A -85,B 0,C 180,E1 -17306.283,E2 -17306.283} C_VEL
LIN {X 0,Y 277.273,Z 347.449,A -85,B 0,C 180,E1 -17310.482,E2 -17310.482} C_VEL
LIN {X 0,Y 277.25,Z 347.565,A -85,B 0,C 180,E1 -17312.164,E2 -17312.164} C_VEL
LIN {X 0,Y 277.534,Z 349.582,A -85,B 0,C 180,E1 -17315.872,E2 -17315.872} C_VEL
LIN {X 0,Y 277.823,Z 351.604,A -85,B 0,C 180,E1 -17319.23,E2 -17319.23} C_VEL
LIN {X 0,Y 278.176,Z 354.079,A -85,B 0,C 180,E1 -17323.012,E2 -17323.012} C_VEL
LIN {X 0,Y 278.324,Z 355.478,A -85,B 0,C 180,E1 -17325.006,E2 -17325.006} C_VEL
LIN {X 0,Y 278.293,Z 357.029,A -85,B 0,C 180,E1 -17327.086,E2 -17327.086} C_VEL
LIN {X 0,Y 277.951,Z 359.977,A -85,B 0,C 180,E1 -17330.793,E2 -17330.793} C_VEL
LIN {X 0,Y 277.452,Z 363.038,A -85,B 0,C 180,E1 -17334.367,E2 -17334.367} C_VEL
LIN {X 0,Y 276.896,Z 366.043,A -85,B 0,C 180,E1 -17337.791,E2 -17337.791} C_VEL
LIN {X 0,Y 276.367,Z 369.121,A -85,B 0,C 180,E1 -17341.108,E2 -17341.108} C_VEL
LIN {X 0,Y 276.141,Z 371.257,A -85,B 0,C 180,E1 -17343.412,E2 -17343.412} C_VEL
LIN {X 0,Y 277.503,Z 376.575,A -85,B 0,C 180,E1 -17343.782,E2 -17343.782} C_VEL
LIN {X 0,Y 280.515,Z 388.199,A -85,B 0,C 180,E1 -17344.791,E2 -17344.791} C_VEL
LIN {X 0,Y 282.293,Z 397.177,A -85,B 0,C 180,E1 -17345.674,E2 -17345.674} C_VEL
LIN {X 0,Y 283.767,Z 408.392,A -85,B 0,C 180,E1 -17346.951,E2 -17346.951} C_VEL
LIN {X 0,Y 284.421,Z 417.115,A -85,B 0,C 180,E1 -17348.09,E2 -17348.09} C_VEL
LIN {X 0,Y 284.398,Z 420.928,A -85,B 0,C 180,E1 -17348.623,E2 -17348.623} C_VEL
LIN {X 0,Y 282.366,Z 432.426,A -85,B 0,C 180,E1 -17350.366,E2 -17350.366} C_VEL
LIN {X 0,Y 280.716,Z 441.217,A -85,B 0,C 180,E1 -17352.06,E2 -17352.06} C_VEL
LIN {X 0,Y 279.547,Z 447.768,A -85,B 0,C 180,E1 -17353.571,E2 -17353.571} C_VEL
LIN {X 0,Y 278.288,Z 454.306,A -85,B 0,C 180,E1 -17355.372,E2 -17355.372} C_VEL
LIN {X 0,Y 277.375,Z 458.807,A -85,B 0,C 180,E1 -17356.818,E2 -17356.818} C_VEL
LIN {X 0,Y 276.441,Z 464.302,A -85,B 0,C 180,E1 -17359.008,E2 -17359.008} C_VEL
LIN {X 0,Y 275.795,Z 468.63,A -85,B 0,C 180,E1 -17361.205,E2 -17361.205} C_VEL
LIN {X 0,Y 275.509,Z 470.999,A -85,B 0,C 180,E1 -17362.672,E2 -17362.672} C_VEL
LIN {X 0,Y 275.267,Z 473.457,A -85,B 0,C 180,E1 -17364.712,E2 -17364.712} C_VEL
LIN {X 0,Y 275.257,Z 475.252,A -85,B 0,C 180,E1 -17367.073,E2 -17367.073} C_VEL
LIN {X 0,Y 275.258,Z 475.842,A -85,B 0,C 180,E1 -17368.537,E2 -17368.537} C_VEL
LIN {X 0,Y 275.257,Z 475.842,A -85,B 0,C 180,E1 -17371.463,E2 -17371.463} C_VEL
LIN {X 0,Y 275.256,Z 475.252,A -85,B 0,C 180,E1 -17372.927,E2 -17372.927} C_VEL
LIN {X 0,Y 275.302,Z 472.799,A -85,B 0,C 180,E1 -17375.861,E2 -17375.861} C_VEL
LIN {X 0,Y 275.619,Z 469.847,A -85,B 0,C 180,E1 -17378.062,E2 -17378.062} C_VEL
LIN {X 0,Y 276.199,Z 465.857,A -85,B 0,C 180,E1 -17380.26,E2 -17380.26} C_VEL
LIN {X 0,Y 277.006,Z 460.723,A -85,B 0,C 180,E1 -17382.454,E2 -17382.454} C_VEL
LIN {X 0,Y 278.04,Z 455.462,A -85,B 0,C 180,E1 -17384.267,E2 -17384.267} C_VEL
LIN {X 0,Y 279.263,Z 449.144,A -85,B 0,C 180,E1 -17386.071,E2 -17386.071} C_VEL
LIN {X 0,Y 280.557,Z 442.521,A -85,B 0,C 180,E1 -17387.649,E2 -17387.649} C_VEL
LIN {X 0,Y 281.948,Z 434.343,A -85,B 0,C 180,E1 -17389.285,E2 -17389.285} C_VEL
LIN {X 0,Y 283.543,Z 425.816,A -85,B 0,C 180,E1 -17390.683,E2 -17390.683} C_VEL
LIN {X 0,Y 284.55,Z 419.574,A -85,B 0,C 180,E1 -17391.555,E2 -17391.555} C_VEL
LIN {X 0,Y 284.004,Z 411.084,A -85,B 0,C 180,E1 -17392.714,E2 -17392.714} C_VEL
LIN {X 0,Y 282.967,Z 401.291,A -85,B 0,C 180,E1 -17393.87,E2 -17393.87} C_VEL
LIN {X 0,Y 281.28,Z 391.749,A -85,B 0,C 180,E1 -17394.866,E2 -17394.866} C_VEL
LIN {X 0,Y 278.895,Z 381.651,A -85,B 0,C 180,E1 -17395.789,E2 -17395.789} C_VEL
LIN {X 0,Y 276.189,Z 371.774,A -85,B 0,C 180,E1 -17396.558,E2 -17396.558} C_VEL
LIN {X 0,Y 276.146,Z 371.266,A -85,B 0,C 180,E1 -17396.587,E2 -17396.587} C_VEL
LIN {X 0,Y 276.663,Z 367.51,A -85,B 0,C 180,E1 -17400.534,E2 -17400.534} C_VEL
LIN {X 0,Y 277.134,Z 364.487,A -85,B 0,C 180,E1 -17403.911,E2 -17403.911} C_VEL
LIN {X 0,Y 277.713,Z 361.465,A -85,B 0,C 180,E1 -17407.399,E2 -17407.399} C_VEL
LIN {X 0,Y 278.174,Z 358.464,A -85,B 0,C 180,E1 -17411.062,E2 -17411.062} C_VEL
LIN {X 0,Y 278.297,Z 356.964,A -85,B 0,C 180,E1 -17412.988,E2 -17412.988} C_VEL
LIN {X 0,Y 278.324,Z 355.467,A -85,B 0,C 180,E1 -17415.005,E2 -17415.005} C_VEL
LIN {X 0,Y 278.02,Z 352.778,A -85,B 0,C 180,E1 -17418.909,E2 -17418.909} C_VEL
LIN {X 0,Y 277.655,Z 350.478,A -85,B 0,C 180,E1 -17422.591,E2 -17422.591} C_VEL
LIN {X 0,Y 277.349,Z 348.137,A -85,B 0,C 180,E1 -17426.742,E2 -17426.742} C_VEL
LIN {X 0,Y 277.25,Z 347.569,A -85,B 0,C 180,E1 -17427.836,E2 -17427.836} C_VEL
LIN {X 0,Y 277.27,Z 347.448,A -85,B 0,C 180,E1 -17431.209,E2 -17431.209} C_VEL
LIN {X 0,Y 277.31,Z 347.442,A -85,B 0,C 180,E1 -17434.478,E2 -17434.478} C_VEL
LIN {X 0,Y 277.267,Z 347.451,A -85,B 0,C 180,E1 -17437.652,E2 -17437.652} C_VEL
LIN {X 0,Y 277.324,Z 347.439,A -85,B 0,C 180,E1 -17440.764,E2 -17440.764} C_VEL
LIN {X 0,Y 277.41,Z 347.431,A -85,B 0,C 180,E1 -17445.324,E2 -17445.324} C_VEL
LIN {X 0,Y 277.507,Z 347.418,A -85,B 0,C 180,E1 -17449.788,E2 -17449.788} C_VEL
LIN {X 0,Y 277.649,Z 347.399,A -85,B 0,C 180,E1 -17452.728,E2 -17452.728} C_VEL
LIN {X 0,Y 277.821,Z 347.375,A -85,B 0,C 180,E1 -17458.55,E2 -17458.55} C_VEL
LIN {X 0,Y 277.82,Z 347.363,A -85,B 0,C 180,E1 -17461.449,E2 -17461.449} C_VEL
LIN {X 0,Y 277.648,Z 347.4,A -85,B 0,C 180,E1 -17467.27,E2 -17467.27} C_VEL
LIN {X 0,Y 277.506,Z 347.413,A -85,B 0,C 180,E1 -17470.21,E2 -17470.21} C_VEL
LIN {X 0,Y 277.433,Z 347.425,A -85,B 0,C 180,E1 -17474.673,E2 -17474.673} C_VEL
LIN {X 0,Y 277.343,Z 347.433,A -85,B 0,C 180,E1 -17479.233,E2 -17479.233} C_VEL
LIN {X 0,Y 277.29,Z 347.443,A -85,B 0,C 180,E1 -17484.157,E2 -17484.157} C_VEL
LIN {X 0,Y 277.326,Z 347.438,A -85,B 0,C 180,E1 -17487.505,E2 -17487.505} C_VEL
LIN {X 0,Y 277.269,Z 347.448,A -85,B 0,C 180,E1 -17490.481,E2 -17490.481} C_VEL
LIN {X 0,Y 277.252,Z 347.448,A -85,B 0,C 180,E1 -17493.894,E2 -17493.894} C_VEL
LIN {X 0,Y 277.288,Z 347.443,A -85,B 0,C 180,E1 -17497.465,E2 -17497.465} C_VEL
LIN {X 0,Y 277.262,Z 347.446,A -85,B 0,C 180,E1 -17501.226,E2 -17501.226} C_VEL
LIN {X 0,Y 277.248,Z 347.447,A -85,B 0,C 180,E1 -17505.215,E2 -17505.215} C_VEL
LIN {X 0,Y 277.284,Z 347.445,A -85,B 0,C 180,E1 -17509.496,E2 -17509.496} C_VEL
LIN {X 0,Y 277.286,Z 347.444,A -85,B 0,C 180,E1 -17512.534,E2 -17512.534} C_VEL
LIN {X 0,Y 277.251,Z 347.451,A -85,B 0,C 180,E1 -17516.105,E2 -17516.105} C_VEL
LIN {X 0,Y 277.258,Z 347.45,A -85,B 0,C 180,E1 -17519.538,E2 -17519.538} C_VEL
LIN {X 0,Y 277.353,Z 347.438,A -85,B 0,C 180,E1 -17523.179,E2 -17523.179} C_VEL
LIN {X 0,Y 278.419,Z 350.389,A -85,B 0,C 180,E1 -17523.394,E2 -17523.394} C_VEL
LIN {X 0,Y 284.773,Z 364,A -85,B 0,C 180,E1 -17524.568,E2 -17524.568} C_VEL
LIN {X 0,Y 289.327,Z 372.282,A -85,B 0,C 180,E1 -17525.489,E2 -17525.489} C_VEL
LIN {X 0,Y 295.668,Z 381.742,A -85,B 0,C 180,E1 -17526.765,E2 -17526.765} C_VEL
LIN {X 0,Y 303.985,Z 392.236,A -85,B 0,C 180,E1 -17528.429,E2 -17528.429} C_VEL
LIN {X 0,Y 312.149,Z 401.635,A -85,B 0,C 180,E1 -17530.11,E2 -17530.11} C_VEL
LIN {X 0,Y 318.547,Z 408.545,A -85,B 0,C 180,E1 -17531.564,E2 -17531.564} C_VEL
LIN {X 0,Y 323.65,Z 413.814,A -85,B 0,C 180,E1 -17532.831,E2 -17532.831} C_VEL
LIN {X 0,Y 330.206,Z 420.123,A -85,B 0,C 180,E1 -17534.589,E2 -17534.589} C_VEL
LIN {X 0,Y 333.667,Z 423.548,A -85,B 0,C 180,E1 -17535.668,E2 -17535.668} C_VEL
LIN {X 0,Y 338.601,Z 427.988,A -85,B 0,C 180,E1 -17537.296,E2 -17537.296} C_VEL
LIN {X 0,Y 343.495,Z 432.182,A -85,B 0,C 180,E1 -17539.136,E2 -17539.136} C_VEL
LIN {X 0,Y 347.065,Z 434.947,A -85,B 0,C 180,E1 -17540.677,E2 -17540.677} C_VEL
LIN {X 0,Y 349.149,Z 437.088,A -85,B 0,C 180,E1 -17541.9,E2 -17541.9} C_VEL
LIN {X 0,Y 351.072,Z 438.801,A -85,B 0,C 180,E1 -17543.101,E2 -17543.101} C_VEL
LIN {X 0,Y 353.044,Z 440.223,A -85,B 0,C 180,E1 -17544.461,E2 -17544.461} C_VEL
LIN {X 0,Y 354.344,Z 440.987,A -85,B 0,C 180,E1 -17545.45,E2 -17545.45} C_VEL
LIN {X 0,Y 355.709,Z 441.544,A -85,B 0,C 180,E1 -17546.602,E2 -17546.602} C_VEL
LIN {X 0,Y 356.757,Z 441.847,A -85,B 0,C 180,E1 -17547.742,E2 -17547.742} C_VEL
LIN {X 0,Y 357.42,Z 441.985,A -85,B 0,C 180,E1 -17548.873,E2 -17548.873} C_VEL
